LIN {X 0,Y 246.753,Z 542.174,A -85,B 0,C 180,E1 -19452.863,E2 -19452.863} C_VEL
LIN {X 0,Y 244.943,Z 545.036,A -85,B 0,C 180,E1 -19455.038,E2 -19455.038} C_VEL
LIN {X 0,Y 243.69,Z 547.692,A -85,B 0,C 180,E1 -19456.783,E2 -19456.783} C_VEL
LIN {X 0,Y 243.644,Z 549.387,A -85,B 0,C 180,E1 -19458.123,E2 -19458.123} C_VEL
LIN {X 0,Y 243.903,Z 549.825,A -85,B 0,C 180,E1 -19458.574,E2 -19458.574} C_VEL
LIN {X 0,Y 249.564,Z 556.197,A -85,B 0,C 180,E1 -19464.321,E2 -19464.321} C_VEL
LIN {X 0,Y 254.169,Z 562.573,A -85,B 0,C 180,E1 -19467.813,E2 -19467.813} C_VEL
LIN {X 0,Y 257.606,Z 568.633,A -85,B 0,C 180,E1 -19470.142,E2 -19470.142} C_VEL
LIN {X 0,Y 261.65,Z 575.949,A -85,B 0,C 180,E1 -19472.607,E2 -19472.607} C_VEL
LIN {X 0,Y 267.284,Z 587.342,A -85,B 0,C 180,E1 -19475.896,E2 -19475.896} C_VEL
LIN {X 0,Y 271.703,Z 597.971,A -85,B 0,C 180,E1 -19478.492,E2 -19478.492} C_VEL
LIN {X 0,Y 273.705,Z 604.625,A -85,B 0,C 180,E1 -19479.839,E2 -19479.839} C_VEL
LIN {X 0,Y 275.017,Z 618.379,A -85,B 0,C 180,E1 -19481.932,E2 -19481.932} C_VEL
LIN {X 0,Y 275.465,Z 630.728,A -85,B 0,C 180,E1 -19483.791,E2 -19483.791} C_VEL
LIN {X 0,Y 274.604,Z 645.683,A -85,B 0,C 180,E1 -19486.014,E2 -19486.014} C_VEL
LIN {X 0,Y 273.727,Z 654.542,A -85,B 0,C 180,E1 -19487.416,E2 -19487.416} C_VEL
LIN {X 0,Y 268.638,Z 668.348,A -85,B 0,C 180,E1 -19489.156,E2 -19489.156} C_VEL
LIN {X 0,Y 263.474,Z 681.321,A -85,B 0,C 180,E1 -19491.185,E2 -19491.185} C_VEL
LIN {X 0,Y 258.614,Z 692.426,A -85,B 0,C 180,E1 -19493.286,E2 -19493.286} C_VEL
LIN {X 0,Y 253.557,Z 703.587,A -85,B 0,C 180,E1 -19495.858,E2 -19495.858} C_VEL
LIN {X 0,Y 249.031,Z 713.236,A -85,B 0,C 180,E1 -19498.529,E2 -19498.529} C_VEL
LIN {X 0,Y 244.437,Z 722.628,A -85,B 0,C 180,E1 -19501.682,E2 -19501.682} C_VEL
LIN {X 0,Y 240.71,Z 730.545,A -85,B 0,C 180,E1 -19504.983,E2 -19504.983} C_VEL
LIN {X 0,Y 237.833,Z 737.107,A -85,B 0,C 180,E1 -19508.325,E2 -19508.325} C_VEL
LIN {X 0,Y 235.644,Z 742.544,A -85,B 0,C 180,E1 -19511.752,E2 -19511.752} C_VEL
LIN {X 0,Y 234.505,Z 745.925,A -85,B 0,C 180,E1 -19514.354,E2 -19514.354} C_VEL
LIN {X 0,Y 233.377,Z 749.429,A -85,B 0,C 180,E1 -19517.833,E2 -19517.833} C_VEL
LIN {X 0,Y 232.962,Z 752.026,A -85,B 0,C 180,E1 -19521.326,E2 -19521.326} C_VEL
LIN {X 0,Y 233.053,Z 753.553,A -85,B 0,C 180,E1 -19524.811,E2 -19524.811} C_VEL
LIN {X 0,Y 233.098,Z 754.168,A -85,B 0,C 180,E1 -19528.274,E2 -19528.274} C_VEL
LIN {X 0,Y 233.218,Z 754.054,A -85,B 0,C 180,E1 -19530.002,E2 -19530.002} C_VEL
LIN {X 0,Y 233.126,Z 753.085,A -85,B 0,C 180,E1 -19533.458,E2 -19533.458} C_VEL
LIN {X 0,Y 233.073,Z 751.097,A -85,B 0,C 180,E1 -19536.929,E2 -19536.929} C_VEL
LIN {X 0,Y 233.202,Z 747.994,A -85,B 0,C 180,E1 -19540.419,E2 -19540.419} C_VEL
LIN {X 0,Y 233.915,Z 743.858,A -85,B 0,C 180,E1 -19543.91,E2 -19543.91} C_VEL
LIN {X 0,Y 235.501,Z 736.962,A -85,B 0,C 180,E1 -19548.263,E2 -19548.263} C_VEL
LIN {X 0,Y 238.22,Z 728.654,A -85,B 0,C 180,E1 -19552.554,E2 -19552.554} C_VEL
LIN {X 0,Y 242.184,Z 720.832,A -85,B 0,C 180,E1 -19556.732,E2 -19556.732} C_VEL
LIN {X 0,Y 247.611,Z 711.66,A -85,B 0,C 180,E1 -19560.725,E2 -19560.725} C_VEL
LIN {X 0,Y 255.156,Z 700.072,A -85,B 0,C 180,E1 -19564.859,E2 -19564.859} C_VEL
LIN {X 0,Y 263.466,Z 688.242,A -85,B 0,C 180,E1 -19568.332,E2 -19568.332} C_VEL
LIN {X 0,Y 273.098,Z 675.378,A -85,B 0,C 180,E1 -19571.437,E2 -19571.437} C_VEL
LIN {X 0,Y 284.184,Z 661.013,A -85,B 0,C 180,E1 -19574.319,E2 -19574.319} C_VEL
LIN {X 0,Y 294.963,Z 646.585,A -85,B 0,C 180,E1 -19577.616,E2 -19577.616} C_VEL
LIN {X 0,Y 295.785,Z 645.371,A -85,B 0,C 180,E1 -19578.296,E2 -19578.296} C_VEL
LIN {X 0,Y 284.508,Z 656.676,A -85,B 0,C 180,E1 -19580.957,E2 -19580.957} C_VEL
LIN {X 0,Y 274.466,Z 666.622,A -85,B 0,C 180,E1 -19583.919,E2 -19583.919} C_VEL
LIN {X 0,Y 265.614,Z 675.208,A -85,B 0,C 180,E1 -19587.152,E2 -19587.152} C_VEL
LIN {X 0,Y 257.876,Z 682.625,A -85,B 0,C 180,E1 -19590.623,E2 -19590.623} C_VEL
LIN {X 0,Y 251.327,Z 688.726,A -85,B 0,C 180,E1 -19594.315,E2 -19594.315} C_VEL
LIN {X 0,Y 245.942,Z 693.539,A -85,B 0,C 180,E1 -19598.194,E2 -19598.194} C_VEL
LIN {X 0,Y 242.458,Z 696.492,A -85,B 0,C 180,E1 -19601.407,E2 -19601.407} C_VEL
LIN {X 0,Y 238.521,Z 699.293,A -85,B 0,C 180,E1 -19606.367,E2 -19606.367} C_VEL
LIN {X 0,Y 236.779,Z 700.073,A -85,B 0,C 180,E1 -19609.742,E2 -19609.742} C_VEL
LIN {X 0,Y 235.445,Z 700.059,A -85,B 0,C 180,E1 -19613.143,E2 -19613.143} C_VEL
LIN {X 0,Y 234.465,Z 699.144,A -85,B 0,C 180,E1 -19616.564,E2 -19616.564} C_VEL
LIN {X 0,Y 234.06,Z 697.294,A -85,B 0,C 180,E1 -19620.001,E2 -19620.001} C_VEL
LIN {X 0,Y 234.205,Z 694.494,A -85,B 0,C 180,E1 -19623.441,E2 -19623.441} C_VEL
LIN {X 0,Y 234.316,Z 690.68,A -85,B 0,C 180,E1 -19626.891,E2 -19626.891} C_VEL
LIN {X 0,Y 234.865,Z 685.837,A -85,B 0,C 180,E1 -19630.344,E2 -19630.344} C_VEL
LIN {X 0,Y 235.755,Z 679.792,A -85,B 0,C 180,E1 -19633.798,E2 -19633.798} C_VEL
LIN {X 0,Y 237.252,Z 672.466,A -85,B 0,C 180,E1 -19637.232,E2 -19637.232} C_VEL
LIN {X 0,Y 239.246,Z 663.732,A -85,B 0,C 180,E1 -19640.642,E2 -19640.642} C_VEL
LIN {X 0,Y 241.824,Z 653.381,A -85,B 0,C 180,E1 -19644.009,E2 -19644.009} C_VEL
LIN {X 0,Y 244.787,Z 641.972,A -85,B 0,C 180,E1 -19647.12,E2 -19647.12} C_VEL
LIN {X 0,Y 247.812,Z 630.51,A -85,B 0,C 180,E1 -19649.757,E2 -19649.757} C_VEL
LIN {X 0,Y 251.044,Z 618.323,A -85,B 0,C 180,E1 -19652.135,E2 -19652.135} C_VEL
LIN {X 0,Y 254.521,Z 604.23,A -85,B 0,C 180,E1 -19654.477,E2 -19654.477} C_VEL
LIN {X 0,Y 257.949,Z 589.052,A -85,B 0,C 180,E1 -19656.585,E2 -19656.585} C_VEL
LIN {X 0,Y 258.395,Z 586.367,A -85,B 0,C 180,E1 -19656.936,E2 -19656.936} C_VEL
LIN {X 0,Y 254.018,Z 573.751,A -85,B 0,C 180,E1 -19659.222,E2 -19659.222} C_VEL
LIN {X 0,Y 248.117,Z 558.525,A -85,B 0,C 180,E1 -19661.873,E2 -19661.873} C_VEL
LIN {X 0,Y 241.376,Z 543.393,A -85,B 0,C 180,E1 -19664.489,E2 -19664.489} C_VEL
LIN {X 0,Y 236.726,Z 534.301,A -85,B 0,C 180,E1 -19666.059,E2 -19666.059} C_VEL
LIN {X 0,Y 235.778,Z 532.761,A -85,B 0,C 180,E1 -19666.392,E2 -19666.392} C_VEL
LIN {X 0,Y 236.767,Z 536.937,A -85,B 0,C 180,E1 -19670.514,E2 -19670.514} C_VEL
LIN {X 0,Y 236.972,Z 538.218,A -85,B 0,C 180,E1 -19671.708,E2 -19671.708} C_VEL
LIN {X 0,Y 238.818,Z 541.601,A -85,B 0,C 180,E1 -19672.353,E2 -19672.353} C_VEL
LIN {X 0,Y 240.695,Z 543.935,A -85,B 0,C 180,E1 -19672.942,E2 -19672.942} C_VEL
LIN {X 0,Y 244.26,Z 549.567,A -85,B 0,C 180,E1 -19674.084,E2 -19674.084} C_VEL
LIN {X 0,Y 248.925,Z 556.937,A -85,B 0,C 180,E1 -19675.567,E2 -19675.567} C_VEL
LIN {X 0,Y 255.974,Z 570.468,A -85,B 0,C 180,E1 -19678.026,E2 -19678.026} C_VEL
LIN {X 0,Y 260.019,Z 580.879,A -85,B 0,C 180,E1 -19679.709,E2 -19679.709} C_VEL
LIN {X 0,Y 264.07,Z 594.759,A -85,B 0,C 180,E1 -19681.87,E2 -19681.87} C_VEL
LIN {X 0,Y 266.896,Z 606.997,A -85,B 0,C 180,E1 -19683.819,E2 -19683.819} C_VEL
LIN {X 0,Y 267.602,Z 611.223,A -85,B 0,C 180,E1 -19684.504,E2 -19684.504} C_VEL
LIN {X 0,Y 264.738,Z 624.004,A -85,B 0,C 180,E1 -19685.909,E2 -19685.909} C_VEL
LIN {X 0,Y 260.749,Z 638.524,A -85,B 0,C 180,E1 -19687.829,E2 -19687.829} C_VEL
LIN {X 0,Y 256.639,Z 651.83,A -85,B 0,C 180,E1 -19689.981,E2 -19689.981} C_VEL
LIN {X 0,Y 252.939,Z 663.185,A -85,B 0,C 180,E1 -19692.202,E2 -19692.202} C_VEL
LIN {X 0,Y 249.018,Z 674.563,A -85,B 0,C 180,E1 -19694.865,E2 -19694.865} C_VEL
LIN {X 0,Y 244.972,Z 685.564,A -85,B 0,C 180,E1 -19697.993,E2 -19697.993} C_VEL
LIN {X 0,Y 242.016,Z 693.828,A -85,B 0,C 180,E1 -19700.878,E2 -19700.878} C_VEL
LIN {X 0,Y 239.165,Z 701.547,A -85,B 0,C 180,E1 -19704.095,E2 -19704.095} C_VEL
LIN {X 0,Y 236.935,Z 708.138,A -85,B 0,C 180,E1 -19707.448,E2 -19707.448} C_VEL
LIN {X 0,Y 234.863,Z 714.656,A -85,B 0,C 180,E1 -19711.713,E2 -19711.713} C_VEL
LIN {X 0,Y 233.843,Z 718.603,A -85,B 0,C 180,E1 -19715.171,E2 -19715.171} C_VEL
LIN {X 0,Y 233.175,Z 721.586,A -85,B 0,C 180,E1 -19718.666,E2 -19718.666} C_VEL
LIN {X 0,Y 232.819,Z 723.564,A -85,B 0,C 180,E1 -19722.197,E2 -19722.197} C_VEL
LIN {X 0,Y 232.769,Z 724.563,A -85,B 0,C 180,E1 -19725.766,E2 -19725.766} C_VEL
LIN {X 0,Y 233.009,Z 724.613,A -85,B 0,C 180,E1 -19729.375,E2 -19729.375} C_VEL
LIN {X 0,Y 233.618,Z 723.592,A -85,B 0,C 180,E1 -19733.02,E2 -19733.02} C_VEL
LIN {X 0,Y 234.77,Z 721.586,A -85,B 0,C 180,E1 -19736.679,E2 -19736.679} C_VEL
LIN {X 0,Y 236.558,Z 718.256,A -85,B 0,C 180,E1 -19740.505,E2 -19740.505} C_VEL
LIN {X 0,Y 238.815,Z 714.066,A -85,B 0,C 180,E1 -19743.994,E2 -19743.994} C_VEL
LIN {X 0,Y 241.917,Z 708.476,A -85,B 0,C 180,E1 -19747.592,E2 -19747.592} C_VEL
LIN {X 0,Y 245.817,Z 701.452,A -85,B 0,C 180,E1 -19751.112,E2 -19751.112} C_VEL
LIN {X 0,Y 250.527,Z 692.801,A -85,B 0,C 180,E1 -19754.53,E2 -19754.53} C_VEL
LIN {X 0,Y 255.281,Z 683.712,A -85,B 0,C 180,E1 -19757.426,E2 -19757.426} C_VEL
LIN {X 0,Y 260.584,Z 672.958,A -85,B 0,C 180,E1 -19760.229,E2 -19760.229} C_VEL
LIN {X 0,Y 266.019,Z 661.133,A -85,B 0,C 180,E1 -19762.735,E2 -19762.735} C_VEL
LIN {X 0,Y 270.921,Z 649.417,A -85,B 0,C 180,E1 -19764.781,E2 -19764.781} C_VEL
LIN {X 0,Y 276.221,Z 635.397,A -85,B 0,C 180,E1 -19766.763,E2 -19766.763} C_VEL
LIN {X 0,Y 280.705,Z 621.712,A -85,B 0,C 180,E1 -19768.345,E2 -19768.345} C_VEL
LIN {X 0,Y 280.523,Z 617.811,A -85,B 0,C 180,E1 -19769.095,E2 -19769.095} C_VEL
LIN {X 0,Y 278.114,Z 605.638,A -85,B 0,C 180,E1 -19771.717,E2 -19771.717} C_VEL
LIN {X 0,Y 275.799,Z 598.13,A -85,B 0,C 180,E1 -19773.516,E2 -19773.516} C_VEL
LIN {X 0,Y 271.396,Z 587.981,A -85,B 0,C 180,E1 -19776.335,E2 -19776.335} C_VEL
LIN {X 0,Y 267.044,Z 579.471,A -85,B 0,C 180,E1 -19778.986,E2 -19778.986} C_VEL
LIN {X 0,Y 263.885,Z 574.325,A -85,B 0,C 180,E1 -19780.857,E2 -19780.857} C_VEL
LIN {X 0,Y 261.135,Z 569.949,A -85,B 0,C 180,E1 -19782.577,E2 -19782.577} C_VEL
LIN {X 0,Y 258.457,Z 565.967,A -85,B 0,C 180,E1 -19784.271,E2 -19784.271} C_VEL
LIN {X 0,Y 255.085,Z 561.378,A -85,B 0,C 180,E1 -19786.557,E2 -19786.557} C_VEL
LIN {X 0,Y 254.143,Z 560.119,A -85,B 0,C 180,E1 -19787.218,E2 -19787.218} C_VEL
LIN {X 0,Y 251.125,Z 556.561,A -85,B 0,C 180,E1 -19789.467,E2 -19789.467} C_VEL
LIN {X 0,Y 250.177,Z 554.992,A -85,B 0,C 180,E1 -19790.296,E2 -19790.296} C_VEL
LIN {X 0,Y 246.659,Z 551.307,A -85,B 0,C 180,E1 -19793.455,E2 -19793.455} C_VEL
LIN {X 0,Y 245.575,Z 549.621,A -85,B 0,C 180,E1 -19794.662,E2 -19794.662} C_VEL
LIN {X 0,Y 240.898,Z 544.483,A -85,B 0,C 180,E1 -19802.194,E2 -19802.194} C_VEL
LIN {X 0,Y 241.02,Z 544.658,A -85,B 0,C 180,E1 -19807.53,E2 -19807.53} C_VEL
LIN {X 0,Y 241.423,Z 545.578,A -85,B 0,C 180,E1 -19811.757,E2 -19811.757} C_VEL
LIN {X 0,Y 242.13,Z 546.869,A -85,B 0,C 180,E1 -19815.142,E2 -19815.142} C_VEL
LIN {X 0,Y 242.607,Z 547.879,A -85,B 0,C 180,E1 -19816.629,E2 -19816.629} C_VEL
LIN {X 0,Y 243.903,Z 549.825,A -85,B 0,C 180,E1 -19818.574,E2 -19818.574} C_VEL
LIN {X 0,Y 244.879,Z 551.629,A -85,B 0,C 180,E1 -19819.87,E2 -19819.87} C_VEL
LIN {X 0,Y 246.399,Z 556.445,A -85,B 0,C 180,E1 -19821.853,E2 -19821.853} C_VEL
LIN {X 0,Y 247.704,Z 560.852,A -85,B 0,C 180,E1 -19823.38,E2 -19823.38} C_VEL
LIN {X 0,Y 249.325,Z 564.702,A -85,B 0,C 180,E1 -19824.955,E2 -19824.955} C_VEL
LIN {X 0,Y 252.237,Z 569.047,A -85,B 0,C 180,E1 -19827.267,E2 -19827.267} C_VEL
LIN {X 0,Y 256.292,Z 576.683,A -85,B 0,C 180,E1 -19830.199,E2 -19830.199} C_VEL
LIN {X 0,Y 258.961,Z 581.967,A -85,B 0,C 180,E1 -19832.009,E2 -19832.009} C_VEL
LIN {X 0,Y 264.002,Z 592.929,A -85,B 0,C 180,E1 -19835.27,E2 -19835.27} C_VEL
LIN {X 0,Y 267.828,Z 603.023,A -85,B 0,C 180,E1 -19837.809,E2 -19837.809} C_VEL
LIN {X 0,Y 269.334,Z 608.443,A -85,B 0,C 180,E1 -19838.979,E2 -19838.979} C_VEL
LIN {X 0,Y 270.277,Z 621.61,A -85,B 0,C 180,E1 -19841.058,E2 -19841.058} C_VEL
LIN {X 0,Y 270.324,Z 634.577,A -85,B 0,C 180,E1 -19843.092,E2 -19843.092} C_VEL
LIN {X 0,Y 269.048,Z 649.765,A -85,B 0,C 180,E1 -19845.451,E2 -19845.451} C_VEL
LIN {X 0,Y 268.079,Z 656.629,A -85,B 0,C 180,E1 -19846.567,E2 -19846.567} C_VEL
LIN {X 0,Y 262.85,Z 669.944,A -85,B 0,C 180,E1 -19848.317,E2 -19848.317} C_VEL
LIN {X 0,Y 257.961,Z 681.592,A -85,B 0,C 180,E1 -19850.193,E2 -19850.193} C_VEL
LIN {X 0,Y 252.932,Z 692.633,A -85,B 0,C 180,E1 -19852.319,E2 -19852.319} C_VEL
LIN {X 0,Y 247.653,Z 703.683,A -85,B 0,C 180,E1 -19854.927,E2 -19854.927} C_VEL
LIN {X 0,Y 242.915,Z 713.226,A -85,B 0,C 180,E1 -19857.642,E2 -19857.642} C_VEL
LIN {X 0,Y 238.131,Z 722.555,A -85,B 0,C 180,E1 -19860.861,E2 -19860.861} C_VEL
LIN {X 0,Y 234.26,Z 730.24,A -85,B 0,C 180,E1 -19864.16,E2 -19864.16} C_VEL
LIN {X 0,Y 231.134,Z 736.895,A -85,B 0,C 180,E1 -19867.664,E2 -19867.664} C_VEL
LIN {X 0,Y 228.788,Z 742.299,A -85,B 0,C 180,E1 -19871.185,E2 -19871.185} C_VEL
LIN {X 0,Y 227.569,Z 745.625,A -85,B 0,C 180,E1 -19873.864,E2 -19873.864} C_VEL
LIN {X 0,Y 226.364,Z 749.09,A -85,B 0,C 180,E1 -19877.45,E2 -19877.45} C_VEL
LIN {X 0,Y 225.891,Z 751.636,A -85,B 0,C 180,E1 -19881.053,E2 -19881.053} C_VEL
LIN {X 0,Y 225.987,Z 753.139,A -85,B 0,C 180,E1 -19884.649,E2 -19884.649} C_VEL
LIN {X 0,Y 226.021,Z 753.704,A -85,B 0,C 180,E1 -19888.22,E2 -19888.22} C_VEL
LIN {X 0,Y 226.134,Z 753.589,A -85,B 0,C 180,E1 -19890.002,E2 -19890.002} C_VEL
LIN {X 0,Y 226.06,Z 752.568,A -85,B 0,C 180,E1 -19893.567,E2 -19893.567} C_VEL
LIN {X 0,Y 226.05,Z 751.42,A -85,B 0,C 180,E1 -19895.8,E2 -19895.8} C_VEL
LIN {X 0,Y 225.986,Z 749.093,A -85,B 0,C 180,E1 -19898.947,E2 -19898.947} C_VEL
LIN {X 0,Y 226.701,Z 744.331,A -85,B 0,C 180,E1 -19903.447,E2 -19903.447} C_VEL
LIN {X 0,Y 227.817,Z 739.299,A -85,B 0,C 180,E1 -19906.998,E2 -19906.998} C_VEL
LIN {X 0,Y 229.659,Z 732.91,A -85,B 0,C 180,E1 -19910.607,E2 -19910.607} C_VEL
LIN {X 0,Y 230.878,Z 729.9,A -85,B 0,C 180,E1 -19912.367,E2 -19912.367} C_VEL
LIN {X 0,Y 234.831,Z 722.594,A -85,B 0,C 180,E1 -19916.676,E2 -19916.676} C_VEL
LIN {X 0,Y 240.264,Z 714.068,A -85,B 0,C 180,E1 -19920.792,E2 -19920.792} C_VEL
LIN {X 0,Y 248.656,Z 702.21,A -85,B 0,C 180,E1 -19925.411,E2 -19925.411} C_VEL
LIN {X 0,Y 258.106,Z 689.925,A -85,B 0,C 180,E1 -19929.279,E2 -19929.279} C_VEL
LIN {X 0,Y 268.204,Z 677.514,A -85,B 0,C 180,E1 -19932.436,E2 -19932.436} C_VEL
LIN {X 0,Y 279.784,Z 663.808,A -85,B 0,C 180,E1 -19935.305,E2 -19935.305} C_VEL
LIN {X 0,Y 287.896,Z 653.936,A -85,B 0,C 180,E1 -19937.692,E2 -19937.692} C_VEL
LIN {X 0,Y 288.836,Z 652.749,A -85,B 0,C 180,E1 -19938.097,E2 -19938.097} C_VEL
LIN {X 0,Y 279.89,Z 660.96,A -85,B 0,C 180,E1 -19940.187,E2 -19940.187} C_VEL
LIN {X 0,Y 269.468,Z 670.219,A -85,B 0,C 180,E1 -19943.141,E2 -19943.141} C_VEL
LIN {X 0,Y 260.249,Z 678.331,A -85,B 0,C 180,E1 -19946.386,E2 -19946.386} C_VEL
LIN {X 0,Y 251.327,Z 685.932,A -85,B 0,C 180,E1 -19950.29,E2 -19950.29} C_VEL
LIN {X 0,Y 244.038,Z 691.945,A -85,B 0,C 180,E1 -19954.407,E2 -19954.407} C_VEL
LIN {X 0,Y 239.597,Z 695.402,A -85,B 0,C 180,E1 -19957.585,E2 -19957.585} C_VEL
LIN {X 0,Y 234.362,Z 699.158,A -85,B 0,C 180,E1 -19962.551,E2 -19962.551} C_VEL
LIN {X 0,Y 230.697,Z 701.035,A -85,B 0,C 180,E1 -19967.688,E2 -19967.688} C_VEL
LIN {X 0,Y 229.157,Z 701.206,A -85,B 0,C 180,E1 -19971.18,E2 -19971.18} C_VEL
LIN {X 0,Y 227.89,Z 700.597,A -85,B 0,C 180,E1 -19974.692,E2 -19974.692} C_VEL
LIN {X 0,Y 227.146,Z 699.046,A -85,B 0,C 180,E1 -19978.228,E2 -19978.228} C_VEL
LIN {X 0,Y 226.978,Z 696.569,A -85,B 0,C 180,E1 -19981.775,E2 -19981.775} C_VEL
LIN {X 0,Y 227.148,Z 694.987,A -85,B 0,C 180,E1 -19983.549,E2 -19983.549} C_VEL
LIN {X 0,Y 227.393,Z 689.847,A -85,B 0,C 180,E1 -19988.031,E2 -19988.031} C_VEL
LIN {X 0,Y 228.051,Z 684.536,A -85,B 0,C 180,E1 -19991.556,E2 -19991.556} C_VEL
LIN {X 0,Y 229.106,Z 678.017,A -85,B 0,C 180,E1 -19995.115,E2 -19995.115} C_VEL
LIN {X 0,Y 231.133,Z 669.112,A -85,B 0,C 180,E1 -19999.08,E2 -19999.08} C_VEL
LIN {X 0,Y 233.46,Z 659.623,A -85,B 0,C 180,E1 -20002.571,E2 -20002.571} C_VEL
LIN {X 0,Y 236.473,Z 648.366,A -85,B 0,C 180,E1 -20006.001,E2 -20006.001} C_VEL
LIN {X 0,Y 239.467,Z 636.847,A -85,B 0,C 180,E1 -20008.964,E2 -20008.964} C_VEL
LIN {X 0,Y 243.428,Z 622.376,A -85,B 0,C 180,E1 -20012.04,E2 -20012.04} C_VEL
LIN {X 0,Y 247.261,Z 607.618,A -85,B 0,C 180,E1 -20014.644,E2 -20014.644} C_VEL
LIN {X 0,Y 250.722,Z 593.093,A -85,B 0,C 180,E1 -20016.793,E2 -20016.793} C_VEL
LIN {X 0,Y 251.718,Z 588.719,A -85,B 0,C 180,E1 -20017.357,E2 -20017.357} C_VEL
LIN {X 0,Y 248.934,Z 579.925,A -85,B 0,C 180,E1 -20019.001,E2 -20019.001} C_VEL
LIN {X 0,Y 243.897,Z 566.294,A -85,B 0,C 180,E1 -20021.511,E2 -20021.511} C_VEL
LIN {X 0,Y 238.559,Z 553.457,A -85,B 0,C 180,E1 -20023.828,E2 -20023.828} C_VEL
LIN {X 0,Y 232.811,Z 541.092,A -85,B 0,C 180,E1 -20026.025,E2 -20026.025} C_VEL
LIN {X 0,Y 231.778,Z 539.224,A -85,B 0,C 180,E1 -20026.382,E2 -20026.382} C_VEL
LIN {X 0,Y 229.341,Z 536.139,A -85,B 0,C 180,E1 -20027.108,E2 -20027.108} C_VEL
LIN {X 0,Y 229.987,Z 538.855,A -85,B 0,C 180,E1 -20029.761,E2 -20029.761} C_VEL
LIN {X 0,Y 231.969,Z 542.273,A -85,B 0,C 180,E1 -20030.504,E2 -20030.504} C_VEL
LIN {X 0,Y 233.725,Z 544.503,A -85,B 0,C 180,E1 -20031.105,E2 -20031.105} C_VEL
LIN {X 0,Y 236.203,Z 548.126,A -85,B 0,C 180,E1 -20031.955,E2 -20031.955} C_VEL
LIN {X 0,Y 240.849,Z 555.572,A -85,B 0,C 180,E1 -20033.567,E2 -20033.567} C_VEL
LIN {X 0,Y 244.842,Z 562.201,A -85,B 0,C 180,E1 -20034.963,E2 -20034.963} C_VEL
LIN {X 0,Y 251.239,Z 574.914,A -85,B 0,C 180,E1 -20037.378,E2 -20037.378} C_VEL
LIN {X 0,Y 254.863,Z 584.868,A -85,B 0,C 180,E1 -20039.066,E2 -20039.066} C_VEL
LIN {X 0,Y 258.336,Z 597.372,A -85,B 0,C 180,E1 -20041.118,E2 -20041.118} C_VEL
LIN {X 0,Y 261.142,Z 610.44,A -85,B 0,C 180,E1 -20043.299,E2 -20043.299} C_VEL
LIN {X 0,Y 261.479,Z 613.997,A -85,B 0,C 180,E1 -20043.861,E2 -20043.861} C_VEL
LIN {X 0,Y 257.585,Z 629.196,A -85,B 0,C 180,E1 -20045.626,E2 -20045.626} C_VEL
LIN {X 0,Y 253.592,Z 642.956,A -85,B 0,C 180,E1 -20047.599,E2 -20047.599} C_VEL
LIN {X 0,Y 249.426,Z 655.715,A -85,B 0,C 180,E1 -20049.807,E2 -20049.807} C_VEL
LIN {X 0,Y 245.089,Z 668.293,A -85,B 0,C 180,E1 -20052.475,E2 -20052.475} C_VEL
LIN {X 0,Y 241.15,Z 678.936,A -85,B 0,C 180,E1 -20055.224,E2 -20055.224} C_VEL
LIN {X 0,Y 237.619,Z 688.069,A -85,B 0,C 180,E1 -20058.05,E2 -20058.05} C_VEL
LIN {X 0,Y 234.303,Z 696.949,A -85,B 0,C 180,E1 -20061.373,E2 -20061.373} C_VEL
LIN {X 0,Y 231.512,Z 704.4,A -85,B 0,C 180,E1 -20064.773,E2 -20064.773} C_VEL
LIN {X 0,Y 228.911,Z 711.887,A -85,B 0,C 180,E1 -20069.119,E2 -20069.119} C_VEL
LIN {X 0,Y 227.22,Z 717.586,A -85,B 0,C 180,E1 -20073.545,E2 -20073.545} C_VEL
LIN {X 0,Y 226.329,Z 720.926,A -85,B 0,C 180,E1 -20077.133,E2 -20077.133} C_VEL
LIN {X 0,Y 225.841,Z 723.338,A -85,B 0,C 180,E1 -20080.759,E2 -20080.759} C_VEL
LIN {X 0,Y 225.719,Z 724.719,A -85,B 0,C 180,E1 -20084.421,E2 -20084.421} C_VEL
LIN {X 0,Y 225.791,Z 725.161,A -85,B 0,C 180,E1 -20088.133,E2 -20088.133} C_VEL
LIN {X 0,Y 226.312,Z 724.602,A -85,B 0,C 180,E1 -20091.877,E2 -20091.877} C_VEL
LIN {X 0,Y 227.584,Z 722.53,A -85,B 0,C 180,E1 -20096.419,E2 -20096.419} C_VEL
LIN {X 0,Y 228.872,Z 720.333,A -85,B 0,C 180,E1 -20099.424,E2 -20099.424} C_VEL
LIN {X 0,Y 231.073,Z 716.46,A -85,B 0,C 180,E1 -20103.191,E2 -20103.191} C_VEL
LIN {X 0,Y 234.065,Z 711.37,A -85,B 0,C 180,E1 -20106.904,E2 -20106.904} C_VEL
LIN {X 0,Y 237.837,Z 704.962,A -85,B 0,C 180,E1 -20110.546,E2 -20110.546} C_VEL
LIN {X 0,Y 242.491,Z 697.048,A -85,B 0,C 180,E1 -20114.07,E2 -20114.07} C_VEL
LIN {X 0,Y 246.907,Z 689.104,A -85,B 0,C 180,E1 -20116.909,E2 -20116.909} C_VEL
LIN {X 0,Y 252.097,Z 679.363,A -85,B 0,C 180,E1 -20119.782,E2 -20119.782} C_VEL
LIN {X 0,Y 257.458,Z 668.759,A -85,B 0,C 180,E1 -20122.335,E2 -20122.335} C_VEL
LIN {X 0,Y 263.296,Z 656.07,A -85,B 0,C 180,E1 -20124.827,E2 -20124.827} C_VEL
LIN {X 0,Y 268.592,Z 643.28,A -85,B 0,C 180,E1 -20126.854,E2 -20126.854} C_VEL
LIN {X 0,Y 273.289,Z 630.509,A -85,B 0,C 180,E1 -20128.516,E2 -20128.516} C_VEL
LIN {X 0,Y 275.539,Z 623.513,A -85,B 0,C 180,E1 -20129.327,E2 -20129.327} C_VEL
LIN {X 0,Y 274.313,Z 614.64,A -85,B 0,C 180,E1 -20131.289,E2 -20131.289} C_VEL
LIN {X 0,Y 272.564,Z 606.596,A -85,B 0,C 180,E1 -20133.176,E2 -20133.176} C_VEL
LIN {X 0,Y 270.258,Z 599.732,A -85,B 0,C 180,E1 -20135.002,E2 -20135.002} C_VEL
LIN {X 0,Y 265.598,Z 588.977,A -85,B 0,C 180,E1 -20138.256,E2 -20138.256} C_VEL
LIN {X 0,Y 261.078,Z 580.613,A -85,B 0,C 180,E1 -20141.255,E2 -20141.255} C_VEL
LIN {X 0,Y 258.197,Z 575.889,A -85,B 0,C 180,E1 -20143.189,E2 -20143.189} C_VEL
LIN {X 0,Y 255.333,Z 571.346,A -85,B 0,C 180,E1 -20145.249,E2 -20145.249} C_VEL
LIN {X 0,Y 252.671,Z 567.345,A -85,B 0,C 180,E1 -20147.232,E2 -20147.232} C_VEL
LIN {X 0,Y 249.307,Z 563.057,A -85,B 0,C 180,E1 -20149.973,E2 -20149.973} C_VEL
LIN {X 0,Y 248.375,Z 561.59,A -85,B 0,C 180,E1 -20150.817,E2 -20150.817} C_VEL
LIN {X 0,Y 245.096,Z 557.788,A -85,B 0,C 180,E1 -20154.033,E2 -20154.033} C_VEL
LIN {X 0,Y 244.274,Z 556.481,A -85,B 0,C 180,E1 -20155.048,E2 -20155.048} C_VEL
LIN {X 0,Y 240.008,Z 551.587,A -85,B 0,C 180,E1 -20162.097,E2 -20162.097} C_VEL
LIN {X 0,Y 238.942,Z 551.538,A -85,B 0,C 180,E1 -20168.456,E2 -20168.456} C_VEL
LIN {X 0,Y 240.291,Z 553.311,A -85,B 0,C 180,E1 -20173.962,E2 -20173.962} C_VEL
LIN {X 0,Y 241.497,Z 554.757,A -85,B 0,C 180,E1 -20176.306,E2 -20176.306} C_VEL
LIN {X 0,Y 247.891,Z 562.589,A -85,B 0,C 180,E1 -20183.717,E2 -20183.717} C_VEL
LIN {X 0,Y 249.325,Z 564.702,A -85,B 0,C 180,E1 -20184.955,E2 -20184.955} C_VEL
LIN {X 0,Y 250.169,Z 566.638,A -85,B 0,C 180,E1 -20185.721,E2 -20185.721} C_VEL
LIN {X 0,Y 251.47,Z 571.825,A -85,B 0,C 180,E1 -20187.067,E2 -20187.067} C_VEL
LIN {X 0,Y 253.45,Z 581.689,A -85,B 0,C 180,E1 -20189.28,E2 -20189.28} C_VEL
LIN {X 0,Y 254.807,Z 584.881,A -85,B 0,C 180,E1 -20190.368,E2 -20190.368} C_VEL
LIN {X 0,Y 258.01,Z 592.18,A -85,B 0,C 180,E1 -20192.762,E2 -20192.762} C_VEL
LIN {X 0,Y 261.56,Z 601.034,A -85,B 0,C 180,E1 -20195.347,E2 -20195.347} C_VEL
LIN {X 0,Y 263.973,Z 608.509,A -85,B 0,C 180,E1 -20197.231,E2 -20197.231} C_VEL
LIN {X 0,Y 265.034,Z 612.903,A -85,B 0,C 180,E1 -20198.193,E2 -20198.193} C_VEL
LIN {X 0,Y 265.543,Z 627.387,A -85,B 0,C 180,E1 -20200.592,E2 -20200.592} C_VEL
LIN {X 0,Y 265.149,Z 638.527,A -85,B 0,C 180,E1 -20202.394,E2 -20202.394} C_VEL
LIN {X 0,Y 263.389,Z 653.939,A -85,B 0,C 180,E1 -20204.927,E2 -20204.927} C_VEL
LIN {X 0,Y 262.515,Z 658.448,A -85,B 0,C 180,E1 -20205.661,E2 -20205.661} C_VEL
LIN {X 0,Y 257.029,Z 671.802,A -85,B 0,C 180,E1 -20207.474,E2 -20207.474} C_VEL
LIN {X 0,Y 251.66,Z 683.813,A -85,B 0,C 180,E1 -20209.515,E2 -20209.515} C_VEL
LIN {X 0,Y 245.66,Z 696.098,A -85,B 0,C 180,E1 -20212.045,E2 -20212.045} C_VEL
LIN {X 0,Y 239.746,Z 707.725,A -85,B 0,C 180,E1 -20215.037,E2 -20215.037} C_VEL
LIN {X 0,Y 234.279,Z 718.041,A -85,B 0,C 180,E1 -20218.336,E2 -20218.336} C_VEL
LIN {X 0,Y 229.717,Z 726.533,A -85,B 0,C 180,E1 -20221.695,E2 -20221.695} C_VEL
LIN {X 0,Y 225.997,Z 733.594,A -85,B 0,C 180,E1 -20225.179,E2 -20225.179} C_VEL
LIN {X 0,Y 223.102,Z 739.506,A -85,B 0,C 180,E1 -20228.763,E2 -20228.763} C_VEL
LIN {X 0,Y 220.944,Z 744.494,A -85,B 0,C 180,E1 -20232.603,E2 -20232.603} C_VEL
LIN {X 0,Y 219.932,Z 747.183,A -85,B 0,C 180,E1 -20235.191,E2 -20235.191} C_VEL
LIN {X 0,Y 219.005,Z 750.111,A -85,B 0,C 180,E1 -20238.901,E2 -20238.901} C_VEL
LIN {X 0,Y 218.8,Z 752.127,A -85,B 0,C 180,E1 -20242.62,E2 -20242.62} C_VEL
LIN {X 0,Y 218.922,Z 752.725,A -85,B 0,C 180,E1 -20244.475,E2 -20244.475} C_VEL
LIN {X 0,Y 218.946,Z 753.239,A -85,B 0,C 180,E1 -20248.163,E2 -20248.163} C_VEL
LIN {X 0,Y 219.053,Z 753.124,A -85,B 0,C 180,E1 -20250.002,E2 -20250.002} C_VEL
LIN {X 0,Y 218.973,Z 752.05,A -85,B 0,C 180,E1 -20253.682,E2 -20253.682} C_VEL
LIN {X 0,Y 218.904,Z 750.002,A -85,B 0,C 180,E1 -20257.38,E2 -20257.38} C_VEL
LIN {X 0,Y 219.107,Z 746.786,A -85,B 0,C 180,E1 -20261.098,E2 -20261.098} C_VEL
LIN {X 0,Y 219.935,Z 742.536,A -85,B 0,C 180,E1 -20264.813,E2 -20264.813} C_VEL
LIN {X 0,Y 221.355,Z 737.054,A -85,B 0,C 180,E1 -20268.514,E2 -20268.514} C_VEL
LIN {X 0,Y 222.906,Z 732.217,A -85,B 0,C 180,E1 -20271.261,E2 -20271.261} C_VEL
LIN {X 0,Y 226.919,Z 725.12,A -85,B 0,C 180,E1 -20276.083,E2 -20276.083} C_VEL
LIN {X 0,Y 231.689,Z 718,A -85,B 0,C 180,E1 -20280.035,E2 -20280.035} C_VEL
LIN {X 0,Y 238.319,Z 709.097,A -85,B 0,C 180,E1 -20284.079,E2 -20284.079} C_VEL
LIN {X 0,Y 248.081,Z 697.027,A -85,B 0,C 180,E1 -20288.555,E2 -20288.555} C_VEL
LIN {X 0,Y 257.851,Z 685.833,A -85,B 0,C 180,E1 -20291.897,E2 -20291.897} C_VEL
LIN {X 0,Y 269.023,Z 673.637,A -85,B 0,C 180,E1 -20294.859,E2 -20294.859} C_VEL
LIN {X 0,Y 275.257,Z 666.908,A -85,B 0,C 180,E1 -20296.266,E2 -20296.266} C_VEL
LIN {X 0,Y 280.265,Z 661.311,A -85,B 0,C 180,E1 -20297.712,E2 -20297.712} C_VEL
LIN {X 0,Y 280.694,Z 660.659,A -85,B 0,C 180,E1 -20298.113,E2 -20298.113} C_VEL
LIN {X 0,Y 268.661,Z 670.474,A -85,B 0,C 180,E1 -20301.111,E2 -20301.111} C_VEL
LIN {X 0,Y 256.733,Z 679.981,A -85,B 0,C 180,E1 -20304.91,E2 -20304.91} C_VEL
LIN {X 0,Y 247.685,Z 686.922,A -85,B 0,C 180,E1 -20308.553,E2 -20308.553} C_VEL
LIN {X 0,Y 240.612,Z 692.174,A -85,B 0,C 180,E1 -20312.139,E2 -20312.139} C_VEL
LIN {X 0,Y 233.292,Z 697.323,A -85,B 0,C 180,E1 -20316.945,E2 -20316.945} C_VEL
LIN {X 0,Y 227.744,Z 700.665,A -85,B 0,C 180,E1 -20322.026,E2 -20322.026} C_VEL
LIN {X 0,Y 224.872,Z 701.945,A -85,B 0,C 180,E1 -20325.667,E2 -20325.667} C_VEL
LIN {X 0,Y 222.995,Z 702.35,A -85,B 0,C 180,E1 -20329.101,E2 -20329.101} C_VEL
LIN {X 0,Y 221.505,Z 701.943,A -85,B 0,C 180,E1 -20332.71,E2 -20332.71} C_VEL
LIN {X 0,Y 220.407,Z 700.709,A -85,B 0,C 180,E1 -20336.344,E2 -20336.344} C_VEL
LIN {X 0,Y 219.926,Z 698.519,A -85,B 0,C 180,E1 -20340.001,E2 -20340.001} C_VEL
LIN {X 0,Y 220.091,Z 695.403,A -85,B 0,C 180,E1 -20343.662,E2 -20343.662} C_VEL
LIN {X 0,Y 220.223,Z 691.3,A -85,B 0,C 180,E1 -20347.335,E2 -20347.335} C_VEL
LIN {X 0,Y 220.826,Z 686.082,A -85,B 0,C 180,E1 -20351.009,E2 -20351.009} C_VEL
LIN {X 0,Y 221.868,Z 679.733,A -85,B 0,C 180,E1 -20354.68,E2 -20354.68} C_VEL
LIN {X 0,Y 223.517,Z 672.061,A -85,B 0,C 180,E1 -20358.327,E2 -20358.327} C_VEL
LIN {X 0,Y 225.796,Z 662.898,A -85,B 0,C 180,E1 -20361.933,E2 -20361.933} C_VEL
LIN {X 0,Y 228.717,Z 652.104,A -85,B 0,C 180,E1 -20365.481,E2 -20365.481} C_VEL
LIN {X 0,Y 231.633,Z 641.292,A -85,B 0,C 180,E1 -20368.48,E2 -20368.48} C_VEL
LIN {X 0,Y 235.285,Z 628.248,A -85,B 0,C 180,E1 -20371.516,E2 -20371.516} C_VEL
LIN {X 0,Y 239.145,Z 614.079,A -85,B 0,C 180,E1 -20374.26,E2 -20374.26} C_VEL
LIN {X 0,Y 242.943,Z 599.386,A -85,B 0,C 180,E1 -20376.631,E2 -20376.631} C_VEL
LIN {X 0,Y 244.953,Z 590.68,A -85,B 0,C 180,E1 -20377.858,E2 -20377.858} C_VEL
LIN {X 0,Y 244.008,Z 586.721,A -85,B 0,C 180,E1 -20378.61,E2 -20378.61} C_VEL
LIN {X 0,Y 238.953,Z 572.48,A -85,B 0,C 180,E1 -20381.376,E2 -20381.376} C_VEL
LIN {X 0,Y 233.296,Z 558.469,A -85,B 0,C 180,E1 -20384.007,E2 -20384.007} C_VEL
LIN {X 0,Y 227.301,Z 545.09,A -85,B 0,C 180,E1 -20386.53,E2 -20386.53} C_VEL
LIN {X 0,Y 223.29,Z 540.218,A -85,B 0,C 180,E1 -20387.714,E2 -20387.714} C_VEL
LIN {X 0,Y 225.696,Z 543.664,A -85,B 0,C 180,E1 -20388.693,E2 -20388.693} C_VEL
LIN {X 0,Y 226.883,Z 545.125,A -85,B 0,C 180,E1 -20389.135,E2 -20389.135} C_VEL
LIN {X 0,Y 229.726,Z 549.174,A -85,B 0,C 180,E1 -20390.189,E2 -20390.189} C_VEL
LIN {X 0,Y 232.781,Z 553.813,A -85,B 0,C 180,E1 -20391.33,E2 -20391.33} C_VEL
LIN {X 0,Y 239.662,Z 565.39,A -85,B 0,C 180,E1 -20393.925,E2 -20393.925} C_VEL
LIN {X 0,Y 245.824,Z 577.972,A -85,B 0,C 180,E1 -20396.468,E2 -20396.468} C_VEL
LIN {X 0,Y 249.148,Z 586.953,A -85,B 0,C 180,E1 -20398.104,E2 -20398.104} C_VEL
LIN {X 0,Y 252.313,Z 598.405,A -85,B 0,C 180,E1 -20400.075,E2 -20400.075} C_VEL
LIN {X 0,Y 255.203,Z 612.621,A -85,B 0,C 180,E1 -20402.554,E2 -20402.554} C_VEL
LIN {X 0,Y 255.479,Z 615.692,A -85,B 0,C 180,E1 -20403.053,E2 -20403.053} C_VEL
LIN {X 0,Y 251.619,Z 630.187,A -85,B 0,C 180,E1 -20404.788,E2 -20404.788} C_VEL
LIN {X 0,Y 247.494,Z 643.862,A -85,B 0,C 180,E1 -20406.795,E2 -20406.795} C_VEL
LIN {X 0,Y 243.518,Z 655.607,A -85,B 0,C 180,E1 -20408.852,E2 -20408.852} C_VEL
LIN {X 0,Y 239.01,Z 668.265,A -85,B 0,C 180,E1 -20411.571,E2 -20411.571} C_VEL
LIN {X 0,Y 234.9,Z 678.967,A -85,B 0,C 180,E1 -20414.377,E2 -20414.377} C_VEL
LIN {X 0,Y 231.19,Z 688.174,A -85,B 0,C 180,E1 -20417.266,E2 -20417.266} C_VEL
LIN {X 0,Y 227.805,Z 696.915,A -85,B 0,C 180,E1 -20420.587,E2 -20420.587} C_VEL
LIN {X 0,Y 224.449,Z 705.442,A -85,B 0,C 180,E1 -20424.608,E2 -20424.608} C_VEL
LIN {X 0,Y 222.25,Z 711.442,A -85,B 0,C 180,E1 -20428.186,E2 -20428.186} C_VEL
LIN {X 0,Y 220.647,Z 716.309,A -85,B 0,C 180,E1 -20431.823,E2 -20431.823} C_VEL
LIN {X 0,Y 219.607,Z 720.145,A -85,B 0,C 180,E1 -20435.507,E2 -20435.507} C_VEL
LIN {X 0,Y 218.916,Z 722.9,A -85,B 0,C 180,E1 -20439.235,E2 -20439.235} C_VEL
LIN {X 0,Y 218.631,Z 724.75,A -85,B 0,C 180,E1 -20443.002,E2 -20443.002} C_VEL
LIN {X 0,Y 218.642,Z 725.547,A -85,B 0,C 180,E1 -20446.813,E2 -20446.813} C_VEL
LIN {X 0,Y 219.027,Z 725.413,A -85,B 0,C 180,E1 -20450.666,E2 -20450.666} C_VEL
LIN {X 0,Y 219.85,Z 724.237,A -85,B 0,C 180,E1 -20454.553,E2 -20454.553} C_VEL
LIN {X 0,Y 221.314,Z 721.988,A -85,B 0,C 180,E1 -20458.444,E2 -20458.444} C_VEL
LIN {X 0,Y 223.424,Z 718.678,A -85,B 0,C 180,E1 -20462.324,E2 -20462.324} C_VEL
LIN {X 0,Y 226.226,Z 714.085,A -85,B 0,C 180,E1 -20466.172,E2 -20466.172} C_VEL
LIN {X 0,Y 229.885,Z 708.216,A -85,B 0,C 180,E1 -20469.939,E2 -20469.939} C_VEL
LIN {X 0,Y 234.421,Z 700.93,A -85,B 0,C 180,E1 -20473.591,E2 -20473.591} C_VEL
LIN {X 0,Y 239.803,Z 692.01,A -85,B 0,C 180,E1 -20477.109,E2 -20477.109} C_VEL
LIN {X 0,Y 245.111,Z 682.641,A -85,B 0,C 180,E1 -20480.081,E2 -20480.081} C_VEL
LIN {X 0,Y 250.179,Z 673.186,A -85,B 0,C 180,E1 -20482.519,E2 -20482.519} C_VEL
LIN {X 0,Y 256.06,Z 661.33,A -85,B 0,C 180,E1 -20485.047,E2 -20485.047} C_VEL
LIN {X 0,Y 261.735,Z 648.737,A -85,B 0,C 180,E1 -20487.23,E2 -20487.23} C_VEL
LIN {X 0,Y 266.583,Z 636.61,A -85,B 0,C 180,E1 -20488.956,E2 -20488.956} C_VEL
LIN {X 0,Y 270.055,Z 626.927,A -85,B 0,C 180,E1 -20490.14,E2 -20490.14} C_VEL
LIN {X 0,Y 270.263,Z 625.372,A -85,B 0,C 180,E1 -20490.39,E2 -20490.39} C_VEL
LIN {X 0,Y 268.957,Z 615.626,A -85,B 0,C 180,E1 -20492.673,E2 -20492.673} C_VEL
LIN {X 0,Y 267.082,Z 607.845,A -85,B 0,C 180,E1 -20494.684,E2 -20494.684} C_VEL
LIN {X 0,Y 264.207,Z 599.998,A -85,B 0,C 180,E1 -20497.034,E2 -20497.034} C_VEL
LIN {X 0,Y 260.964,Z 592.557,A -85,B 0,C 180,E1 -20499.506,E2 -20499.506} C_VEL
LIN {X 0,Y 256.983,Z 584.958,A -85,B 0,C 180,E1 -20502.441,E2 -20502.441} C_VEL
LIN {X 0,Y 255.136,Z 581.668,A -85,B 0,C 180,E1 -20503.856,E2 -20503.856} C_VEL
LIN {X 0,Y 252.636,Z 577.492,A -85,B 0,C 180,E1 -20505.808,E2 -20505.808} C_VEL
LIN {X 0,Y 249.952,Z 573.179,A -85,B 0,C 180,E1 -20508.084,E2 -20508.084} C_VEL
LIN {X 0,Y 247.251,Z 569.444,A -85,B 0,C 180,E1 -20510.489,E2 -20510.489} C_VEL
LIN {X 0,Y 246.357,Z 568.089,A -85,B 0,C 180,E1 -20511.386,E2 -20511.386} C_VEL
LIN {X 0,Y 243.374,Z 564.121,A -85,B 0,C 180,E1 -20514.718,E2 -20514.718} C_VEL
LIN {X 0,Y 242.813,Z 563.297,A -85,B 0,C 180,E1 -20515.434,E2 -20515.434} C_VEL
LIN {X 0,Y 239.096,Z 558.659,A -85,B 0,C 180,E1 -20522.063,E2 -20522.063} C_VEL
LIN {X 0,Y 238.049,Z 558.597,A -85,B 0,C 180,E1 -20528.488,E2 -20528.488} C_VEL
LIN {X 0,Y 239.341,Z 560.339,A -85,B 0,C 180,E1 -20533.856,E2 -20533.856} C_VEL
LIN {X 0,Y 240.411,Z 561.673,A -85,B 0,C 180,E1 -20536.018,E2 -20536.018} C_VEL
LIN {X 0,Y 246.327,Z 569.299,A -85,B 0,C 180,E1 -20543.319,E2 -20543.319} C_VEL
LIN {X 0,Y 250.066,Z 575.126,A -85,B 0,C 180,E1 -20546.585,E2 -20546.585} C_VEL
LIN {X 0,Y 253.863,Z 582.927,A -85,B 0,C 180,E1 -20549.659,E2 -20549.659} C_VEL
LIN {X 0,Y 254.807,Z 584.881,A -85,B 0,C 180,E1 -20550.368,E2 -20550.368} C_VEL
LIN {X 0,Y 255.75,Z 586.912,A -85,B 0,C 180,E1 -20551.086,E2 -20551.086} C_VEL
LIN {X 0,Y 256.682,Z 590.955,A -85,B 0,C 180,E1 -20552.023,E2 -20552.023} C_VEL
LIN {X 0,Y 257.83,Z 605.245,A -85,B 0,C 180,E1 -20554.493,E2 -20554.493} C_VEL
LIN {X 0,Y 258.37,Z 608.018,A -85,B 0,C 180,E1 -20555.133,E2 -20555.133} C_VEL
LIN {X 0,Y 259.934,Z 613.276,A -85,B 0,C 180,E1 -20556.5,E2 -20556.5} C_VEL
LIN {X 0,Y 260.661,Z 617.149,A -85,B 0,C 180,E1 -20557.386,E2 -20557.386} C_VEL
LIN {X 0,Y 260.768,Z 629.988,A -85,B 0,C 180,E1 -20559.585,E2 -20559.585} C_VEL
LIN {X 0,Y 260.08,Z 641.209,A -85,B 0,C 180,E1 -20561.483,E2 -20561.483} C_VEL
LIN {X 0,Y 258.021,Z 656.063,A -85,B 0,C 180,E1 -20564.015,E2 -20564.015} C_VEL
LIN {X 0,Y 257.449,Z 659.071,A -85,B 0,C 180,E1 -20564.563,E2 -20564.563} C_VEL
LIN {X 0,Y 252.07,Z 671.732,A -85,B 0,C 180,E1 -20566.308,E2 -20566.308} C_VEL
LIN {X 0,Y 246.287,Z 684.121,A -85,B 0,C 180,E1 -20568.439,E2 -20568.439} C_VEL
LIN {X 0,Y 240.085,Z 696.278,A -85,B 0,C 180,E1 -20570.999,E2 -20570.999} C_VEL
LIN {X 0,Y 233.753,Z 708.055,A -85,B 0,C 180,E1 -20574.109,E2 -20574.109} C_VEL
LIN {X 0,Y 228.189,Z 717.998,A -85,B 0,C 180,E1 -20577.388,E2 -20577.388} C_VEL
LIN {X 0,Y 223.392,Z 726.436,A -85,B 0,C 180,E1 -20580.817,E2 -20580.817} C_VEL
LIN {X 0,Y 219.461,Z 733.433,A -85,B 0,C 180,E1 -20584.387,E2 -20584.387} C_VEL
LIN {X 0,Y 216.395,Z 739.273,A -85,B 0,C 180,E1 -20588.071,E2 -20588.071} C_VEL
LIN {X 0,Y 213.953,Z 744.517,A -85,B 0,C 180,E1 -20592.286,E2 -20592.286} C_VEL
LIN {X 0,Y 212.383,Z 748.427,A -85,B 0,C 180,E1 -20596.609,E2 -20596.609} C_VEL
LIN {X 0,Y 211.744,Z 750.857,A -85,B 0,C 180,E1 -20600.449,E2 -20600.449} C_VEL
LIN {X 0,Y 211.847,Z 752.345,A -85,B 0,C 180,E1 -20604.402,E2 -20604.402} C_VEL
LIN {X 0,Y 211.872,Z 752.773,A -85,B 0,C 180,E1 -20608.101,E2 -20608.101} C_VEL
LIN {X 0,Y 211.974,Z 752.657,A -85,B 0,C 180,E1 -20610.002,E2 -20610.002} C_VEL
LIN {X 0,Y 211.888,Z 751.529,A -85,B 0,C 180,E1 -20613.806,E2 -20613.806} C_VEL
LIN {X 0,Y 211.907,Z 750.582,A -85,B 0,C 180,E1 -20615.76,E2 -20615.76} C_VEL
LIN {X 0,Y 211.844,Z 747.935,A -85,B 0,C 180,E1 -20619.55,E2 -20619.55} C_VEL
LIN {X 0,Y 212.459,Z 744.151,A -85,B 0,C 180,E1 -20623.391,E2 -20623.391} C_VEL
LIN {X 0,Y 213.775,Z 738.76,A -85,B 0,C 180,E1 -20627.564,E2 -20627.564} C_VEL
LIN {X 0,Y 215.556,Z 733.109,A -85,B 0,C 180,E1 -20631.019,E2 -20631.019} C_VEL
LIN {X 0,Y 220.242,Z 725.537,A -85,B 0,C 180,E1 -20636.687,E2 -20636.687} C_VEL
LIN {X 0,Y 225.525,Z 718.34,A -85,B 0,C 180,E1 -20640.945,E2 -20640.945} C_VEL
LIN {X 0,Y 233.949,Z 708.177,A -85,B 0,C 180,E1 -20645.798,E2 -20645.798} C_VEL
LIN {X 0,Y 244.573,Z 696.38,A -85,B 0,C 180,E1 -20650.284,E2 -20650.284} C_VEL
LIN {X 0,Y 257.231,Z 683.345,A -85,B 0,C 180,E1 -20654.165,E2 -20654.165} C_VEL
LIN {X 0,Y 271.202,Z 669.59,A -85,B 0,C 180,E1 -20657.362,E2 -20657.362} C_VEL
LIN {X 0,Y 272.562,Z 668.183,A -85,B 0,C 180,E1 -20657.722,E2 -20657.722} C_VEL
LIN {X 0,Y 273.093,Z 667.543,A -85,B 0,C 180,E1 -20658.003,E2 -20658.003} C_VEL
LIN {X 0,Y 261.72,Z 675.863,A -85,B 0,C 180,E1 -20660.873,E2 -20660.873} C_VEL
LIN {X 0,Y 250.21,Z 684.018,A -85,B 0,C 180,E1 -20664.546,E2 -20664.546} C_VEL
LIN {X 0,Y 240.818,Z 690.453,A -85,B 0,C 180,E1 -20668.312,E2 -20668.312} C_VEL
LIN {X 0,Y 234.706,Z 694.501,A -85,B 0,C 180,E1 -20671.374,E2 -20671.374} C_VEL
LIN {X 0,Y 226.993,Z 699.151,A -85,B 0,C 180,E1 -20676.266,E2 -20676.266} C_VEL
LIN {X 0,Y 222.908,Z 701.349,A -85,B 0,C 180,E1 -20679.708,E2 -20679.708} C_VEL
LIN {X 0,Y 219.564,Z 702.799,A -85,B 0,C 180,E1 -20683.258,E2 -20683.258} C_VEL
LIN {X 0,Y 217.025,Z 703.422,A -85,B 0,C 180,E1 -20686.899,E2 -20686.899} C_VEL
LIN {X 0,Y 215.302,Z 703.255,A -85,B 0,C 180,E1 -20690.607,E2 -20690.607} C_VEL
LIN {X 0,Y 213.896,Z 702.249,A -85,B 0,C 180,E1 -20694.344,E2 -20694.344} C_VEL
LIN {X 0,Y 213.035,Z 700.39,A -85,B 0,C 180,E1 -20698.11,E2 -20698.11} C_VEL
LIN {X 0,Y 212.866,Z 697.55,A -85,B 0,C 180,E1 -20701.893,E2 -20701.893} C_VEL
LIN {X 0,Y 213.015,Z 695.774,A -85,B 0,C 180,E1 -20703.784,E2 -20703.784} C_VEL
LIN {X 0,Y 213.175,Z 691.549,A -85,B 0,C 180,E1 -20707.579,E2 -20707.579} C_VEL
LIN {X 0,Y 213.834,Z 686.143,A -85,B 0,C 180,E1 -20711.374,E2 -20711.374} C_VEL
LIN {X 0,Y 214.917,Z 679.577,A -85,B 0,C 180,E1 -20715.166,E2 -20715.166} C_VEL
LIN {X 0,Y 216.709,Z 671.742,A -85,B 0,C 180,E1 -20718.924,E2 -20718.924} C_VEL
LIN {X 0,Y 219.109,Z 662.41,A -85,B 0,C 180,E1 -20722.639,E2 -20722.639} C_VEL
LIN {X 0,Y 222.2,Z 651.357,A -85,B 0,C 180,E1 -20726.284,E2 -20726.284} C_VEL
LIN {X 0,Y 225.45,Z 639.54,A -85,B 0,C 180,E1 -20729.552,E2 -20729.552} C_VEL
LIN {X 0,Y 229.092,Z 626.924,A -85,B 0,C 180,E1 -20732.471,E2 -20732.471} C_VEL
LIN {X 0,Y 232.739,Z 613.919,A -85,B 0,C 180,E1 -20735.012,E2 -20735.012} C_VEL
LIN {X 0,Y 236.732,Z 598.821,A -85,B 0,C 180,E1 -20737.489,E2 -20737.489} C_VEL
LIN {X 0,Y 238.36,Z 591.678,A -85,B 0,C 180,E1 -20738.526,E2 -20738.526} C_VEL
LIN {X 0,Y 233.741,Z 578.259,A -85,B 0,C 180,E1 -20741.261,E2 -20741.261} C_VEL
LIN {X 0,Y 228.826,Z 565.375,A -85,B 0,C 180,E1 -20743.798,E2 -20743.798} C_VEL
LIN {X 0,Y 223.039,Z 551.888,A -85,B 0,C 180,E1 -20746.448,E2 -20746.448} C_VEL
LIN {X 0,Y 220.859,Z 547.973,A -85,B 0,C 180,E1 -20747.273,E2 -20747.273} C_VEL
LIN {X 0,Y 221.925,Z 548.69,A -85,B 0,C 180,E1 -20747.74,E2 -20747.74} C_VEL
LIN {X 0,Y 223.634,Z 550.892,A -85,B 0,C 180,E1 -20748.419,E2 -20748.419} C_VEL
LIN {X 0,Y 227.515,Z 556.952,A -85,B 0,C 180,E1 -20750.002,E2 -20750.002} C_VEL
LIN {X 0,Y 230.097,Z 560.967,A -85,B 0,C 180,E1 -20751.034,E2 -20751.034} C_VEL
LIN {X 0,Y 235.958,Z 571.334,A -85,B 0,C 180,E1 -20753.475,E2 -20753.475} C_VEL
LIN {X 0,Y 241.543,Z 583.511,A -85,B 0,C 180,E1 -20756.024,E2 -20756.024} C_VEL
LIN {X 0,Y 244.839,Z 593.645,A -85,B 0,C 180,E1 -20757.924,E2 -20757.924} C_VEL
LIN {X 0,Y 247.634,Z 605.793,A -85,B 0,C 180,E1 -20760.113,E2 -20760.113} C_VEL
LIN {X 0,Y 249.525,Z 616.31,A -85,B 0,C 180,E1 -20762.043,E2 -20762.043} C_VEL
LIN {X 0,Y 249.33,Z 618.366,A -85,B 0,C 180,E1 -20762.333,E2 -20762.333} C_VEL
LIN {X 0,Y 245.325,Z 632.541,A -85,B 0,C 180,E1 -20764.094,E2 -20764.094} C_VEL
LIN {X 0,Y 241.076,Z 645.887,A -85,B 0,C 180,E1 -20766.139,E2 -20766.139} C_VEL
LIN {X 0,Y 236.995,Z 657.369,A -85,B 0,C 180,E1 -20768.241,E2 -20768.241} C_VEL
LIN {X 0,Y 232.35,Z 669.831,A -85,B 0,C 180,E1 -20771.023,E2 -20771.023} C_VEL
LIN {X 0,Y 228.133,Z 680.425,A -85,B 0,C 180,E1 -20773.902,E2 -20773.902} C_VEL
LIN {X 0,Y 223.839,Z 690.668,A -85,B 0,C 180,E1 -20777.302,E2 -20777.302} C_VEL
LIN {X 0,Y 220.332,Z 699.247,A -85,B 0,C 180,E1 -20780.821,E2 -20780.821} C_VEL
LIN {X 0,Y 217.402,Z 706.452,A -85,B 0,C 180,E1 -20784.433,E2 -20784.433} C_VEL
LIN {X 0,Y 215.142,Z 712.393,A -85,B 0,C 180,E1 -20788.126,E2 -20788.126} C_VEL
LIN {X 0,Y 213.544,Z 717.133,A -85,B 0,C 180,E1 -20791.884,E2 -20791.884} C_VEL
LIN {X 0,Y 212.495,Z 720.885,A -85,B 0,C 180,E1 -20795.692,E2 -20795.692} C_VEL
LIN {X 0,Y 211.779,Z 723.559,A -85,B 0,C 180,E1 -20799.549,E2 -20799.549} C_VEL
LIN {X 0,Y 211.542,Z 725.295,A -85,B 0,C 180,E1 -20803.446,E2 -20803.446} C_VEL
LIN {X 0,Y 211.584,Z 726.042,A -85,B 0,C 180,E1 -20807.392,E2 -20807.392} C_VEL
LIN {X 0,Y 212.169,Z 725.671,A -85,B 0,C 180,E1 -20811.951,E2 -20811.951} C_VEL
LIN {X 0,Y 213.012,Z 724.564,A -85,B 0,C 180,E1 -20815.396,E2 -20815.396} C_VEL
LIN {X 0,Y 214.645,Z 722.197,A -85,B 0,C 180,E1 -20819.413,E2 -20819.413} C_VEL
LIN {X 0,Y 216.959,Z 718.762,A -85,B 0,C 180,E1 -20823.411,E2 -20823.411} C_VEL
LIN {X 0,Y 220.077,Z 714.101,A -85,B 0,C 180,E1 -20827.352,E2 -20827.352} C_VEL
LIN {X 0,Y 224.035,Z 708.092,A -85,B 0,C 180,E1 -20831.203,E2 -20831.203} C_VEL
LIN {X 0,Y 228.912,Z 700.662,A -85,B 0,C 180,E1 -20834.918,E2 -20834.918} C_VEL
LIN {X 0,Y 233.883,Z 692.857,A -85,B 0,C 180,E1 -20838.046,E2 -20838.046} C_VEL
LIN {X 0,Y 239.406,Z 683.527,A -85,B 0,C 180,E1 -20841.068,E2 -20841.068} C_VEL
LIN {X 0,Y 244.677,Z 674.16,A -85,B 0,C 180,E1 -20843.535,E2 -20843.535} C_VEL
LIN {X 0,Y 250.712,Z 662.519,A -85,B 0,C 180,E1 -20846.068,E2 -20846.068} C_VEL
LIN {X 0,Y 256.367,Z 650.567,A -85,B 0,C 180,E1 -20848.189,E2 -20848.189} C_VEL
LIN {X 0,Y 261.641,Z 637.919,A -85,B 0,C 180,E1 -20850.024,E2 -20850.024} C_VEL
LIN {X 0,Y 264.89,Z 629.254,A -85,B 0,C 180,E1 -20851.105,E2 -20851.105} C_VEL
LIN {X 0,Y 264.861,Z 625.925,A -85,B 0,C 180,E1 -20851.842,E2 -20851.842} C_VEL
LIN {X 0,Y 263.769,Z 617.586,A -85,B 0,C 180,E1 -20853.919,E2 -20853.919} C_VEL
LIN {X 0,Y 262.116,Z 610.844,A -85,B 0,C 180,E1 -20855.822,E2 -20855.822} C_VEL
LIN {X 0,Y 258.681,Z 601.345,A -85,B 0,C 180,E1 -20858.9,E2 -20858.9} C_VEL
LIN {X 0,Y 255.502,Z 594.218,A -85,B 0,C 180,E1 -20861.558,E2 -20861.558} C_VEL
LIN {X 0,Y 252.839,Z 588.66,A -85,B 0,C 180,E1 -20863.861,E2 -20863.861} C_VEL
LIN {X 0,Y 250.527,Z 584.617,A -85,B 0,C 180,E1 -20865.79,E2 -20865.79} C_VEL
LIN {X 0,Y 247.433,Z 579.468,A -85,B 0,C 180,E1 -20868.635,E2 -20868.635} C_VEL
LIN {X 0,Y 244.881,Z 575.449,A -85,B 0,C 180,E1 -20871.229,E2 -20871.229} C_VEL
LIN {X 0,Y 241.14,Z 570.095,A -85,B 0,C 180,E1 -20875.821,E2 -20875.821} C_VEL
LIN {X 0,Y 237.988,Z 565.721,A -85,B 0,C 180,E1 -20882.072,E2 -20882.072} C_VEL
LIN {X 0,Y 236.974,Z 565.449,A -85,B 0,C 180,E1 -20886.812,E2 -20886.812} C_VEL
LIN {X 0,Y 237.587,Z 566.577,A -85,B 0,C 180,E1 -20891.95,E2 -20891.95} C_VEL
LIN {X 0,Y 239.066,Z 568.385,A -85,B 0,C 180,E1 -20895.56,E2 -20895.56} C_VEL
LIN {X 0,Y 244.59,Z 575.977,A -85,B 0,C 180,E1 -20902.913,E2 -20902.913} C_VEL
LIN {X 0,Y 247.827,Z 581.424,A -85,B 0,C 180,E1 -20906.018,E2 -20906.018} C_VEL
LIN {X 0,Y 251.066,Z 588.752,A -85,B 0,C 180,E1 -20908.987,E2 -20908.987} C_VEL
LIN {X 0,Y 253.221,Z 593.799,A -85,B 0,C 180,E1 -20910.788,E2 -20910.788} C_VEL
LIN {X 0,Y 257.668,Z 605.495,A -85,B 0,C 180,E1 -20914.468,E2 -20914.468} C_VEL
LIN {X 0,Y 258.37,Z 608.018,A -85,B 0,C 180,E1 -20915.133,E2 -20915.133} C_VEL
LIN {X 0,Y 258.891,Z 610.78,A -85,B 0,C 180,E1 -20915.744,E2 -20915.744} C_VEL
LIN {X 0,Y 258.918,Z 615.598,A -85,B 0,C 180,E1 -20916.51,E2 -20916.51} C_VEL
LIN {X 0,Y 258.275,Z 620.794,A -85,B 0,C 180,E1 -20917.151,E2 -20917.151} C_VEL
LIN {X 0,Y 256.322,Z 631.448,A -85,B 0,C 180,E1 -20918.43,E2 -20918.43} C_VEL
LIN {X 0,Y 255.902,Z 634.755,A -85,B 0,C 180,E1 -20918.952,E2 -20918.952} C_VEL
LIN {X 0,Y 254.934,Z 644.582,A -85,B 0,C 180,E1 -20920.672,E2 -20920.672} C_VEL
LIN {X 0,Y 252.521,Z 658.841,A -85,B 0,C 180,E1 -20923.214,E2 -20923.214} C_VEL
LIN {X 0,Y 252.123,Z 660.695,A -85,B 0,C 180,E1 -20923.555,E2 -20923.555} C_VEL
LIN {X 0,Y 245.769,Z 674.674,A -85,B 0,C 180,E1 -20925.581,E2 -20925.581} C_VEL
LIN {X 0,Y 240.039,Z 686.28,A -85,B 0,C 180,E1 -20927.672,E2 -20927.672} C_VEL
LIN {X 0,Y 233.7,Z 698.075,A -85,B 0,C 180,E1 -20930.282,E2 -20930.282} C_VEL
LIN {X 0,Y 227.832,Z 708.396,A -85,B 0,C 180,E1 -20933.135,E2 -20933.135} C_VEL
LIN {X 0,Y 222.194,Z 717.976,A -85,B 0,C 180,E1 -20936.394,E2 -20936.394} C_VEL
LIN {X 0,Y 217.114,Z 726.323,A -85,B 0,C 180,E1 -20939.888,E2 -20939.888} C_VEL
LIN {X 0,Y 212.972,Z 733.273,A -85,B 0,C 180,E1 -20943.548,E2 -20943.548} C_VEL
LIN {X 0,Y 209.705,Z 739.042,A -85,B 0,C 180,E1 -20947.333,E2 -20947.333} C_VEL
LIN {X 0,Y 206.942,Z 744.507,A -85,B 0,C 180,E1 -20951.971,E2 -20951.971} C_VEL
LIN {X 0,Y 205.386,Z 748.099,A -85,B 0,C 180,E1 -20956.144,E2 -20956.144} C_VEL
LIN {X 0,Y 204.667,Z 750.469,A -85,B 0,C 180,E1 -20960.116,E2 -20960.116} C_VEL
LIN {X 0,Y 204.748,Z 752.016,A -85,B 0,C 180,E1 -20964.512,E2 -20964.512} C_VEL
LIN {X 0,Y 204.8,Z 752.307,A -85,B 0,C 180,E1 -20968.036,E2 -20968.036} C_VEL
LIN {X 0,Y 204.897,Z 752.175,A -85,B 0,C 180,E1 -20970.002,E2 -20970.002} C_VEL
LIN {X 0,Y 204.807,Z 751.007,A -85,B 0,C 180,E1 -20973.937,E2 -20973.937} C_VEL
LIN {X 0,Y 204.814,Z 750.058,A -85,B 0,C 180,E1 -20975.911,E2 -20975.911} C_VEL
LIN {X 0,Y 204.789,Z 747.353,A -85,B 0,C 180,E1 -20979.882,E2 -20979.882} C_VEL
LIN {X 0,Y 205.48,Z 743.507,A -85,B 0,C 180,E1 -20983.854,E2 -20983.854} C_VEL
LIN {X 0,Y 206.808,Z 738.426,A -85,B 0,C 180,E1 -20987.915,E2 -20987.915} C_VEL
LIN {X 0,Y 208.822,Z 732.74,A -85,B 0,C 180,E1 -20991.73,E2 -20991.73} C_VEL
LIN {X 0,Y 213.566,Z 725.896,A -85,B 0,C 180,E1 -20997.315,E2 -20997.315} C_VEL
LIN {X 0,Y 219.418,Z 718.73,A -85,B 0,C 180,E1 -21001.906,E2 -21001.906} C_VEL
LIN {X 0,Y 228.19,Z 709.176,A -85,B 0,C 180,E1 -21006.797,E2 -21006.797} C_VEL
LIN {X 0,Y 239.341,Z 697.933,A -85,B 0,C 180,E1 -21011.354,E2 -21011.354} C_VEL
LIN {X 0,Y 253.602,Z 684.528,A -85,B 0,C 180,E1 -21015.531,E2 -21015.531} C_VEL
LIN {X 0,Y 264.781,Z 674.407,A -85,B 0,C 180,E1 -21018.006,E2 -21018.006} C_VEL
LIN {X 0,Y 252.602,Z 682.328,A -85,B 0,C 180,E1 -21021.245,E2 -21021.245} C_VEL
LIN {X 0,Y 240.564,Z 689.877,A -85,B 0,C 180,E1 -21025.273,E2 -21025.273} C_VEL
LIN {X 0,Y 231.91,Z 695.007,A -85,B 0,C 180,E1 -21028.991,E2 -21028.991} C_VEL
LIN {X 0,Y 223.252,Z 699.776,A -85,B 0,C 180,E1 -21033.851,E2 -21033.851} C_VEL
LIN {X 0,Y 216.462,Z 702.992,A -85,B 0,C 180,E1 -21039.076,E2 -21039.076} C_VEL
LIN {X 0,Y 211.471,Z 704.489,A -85,B 0,C 180,E1 -21044.582,E2 -21044.582} C_VEL
LIN {X 0,Y 209.19,Z 704.5,A -85,B 0,C 180,E1 -21048.372,E2 -21048.372} C_VEL
LIN {X 0,Y 207.561,Z 703.748,A -85,B 0,C 180,E1 -21052.217,E2 -21052.217} C_VEL
LIN {X 0,Y 206.31,Z 702.12,A -85,B 0,C 180,E1 -21056.094,E2 -21056.094} C_VEL
LIN {X 0,Y 205.801,Z 699.619,A -85,B 0,C 180,E1 -21060.001,E2 -21060.001} C_VEL
LIN {X 0,Y 205.925,Z 696.133,A -85,B 0,C 180,E1 -21063.915,E2 -21063.915} C_VEL
LIN {X 0,Y 206.113,Z 691.676,A -85,B 0,C 180,E1 -21067.84,E2 -21067.84} C_VEL
LIN {X 0,Y 206.817,Z 686.19,A -85,B 0,C 180,E1 -21071.765,E2 -21071.765} C_VEL
LIN {X 0,Y 207.99,Z 679.389,A -85,B 0,C 180,E1 -21075.684,E2 -21075.684} C_VEL
LIN {X 0,Y 209.924,Z 671.309,A -85,B 0,C 180,E1 -21079.561,E2 -21079.561} C_VEL
LIN {X 0,Y 212.452,Z 661.751,A -85,B 0,C 180,E1 -21083.39,E2 -21083.39} C_VEL
LIN {X 0,Y 215.716,Z 650.504,A -85,B 0,C 180,E1 -21087.138,E2 -21087.138} C_VEL
LIN {X 0,Y 219.084,Z 638.701,A -85,B 0,C 180,E1 -21090.425,E2 -21090.425} C_VEL
LIN {X 0,Y 223.276,Z 624.487,A -85,B 0,C 180,E1 -21093.696,E2 -21093.696} C_VEL
LIN {X 0,Y 227.254,Z 610.509,A -85,B 0,C 180,E1 -21096.376,E2 -21096.376} C_VEL
LIN {X 0,Y 231.291,Z 595.256,A -85,B 0,C 180,E1 -21098.809,E2 -21098.809} C_VEL
LIN {X 0,Y 231.646,Z 593.789,A -85,B 0,C 180,E1 -21099.017,E2 -21099.017} C_VEL
LIN {X 0,Y 227.361,Z 580.852,A -85,B 0,C 180,E1 -21101.754,E2 -21101.754} C_VEL
LIN {X 0,Y 222.576,Z 568.039,A -85,B 0,C 180,E1 -21104.404,E2 -21104.404} C_VEL
LIN {X 0,Y 217.656,Z 556.451,A -85,B 0,C 180,E1 -21106.793,E2 -21106.793} C_VEL
LIN {X 0,Y 218.386,Z 556.762,A -85,B 0,C 180,E1 -21107.066,E2 -21107.066} C_VEL
LIN {X 0,Y 220.304,Z 556.546,A -85,B 0,C 180,E1 -21107.699,E2 -21107.699} C_VEL
LIN {X 0,Y 226.268,Z 566.238,A -85,B 0,C 180,E1 -21110.33,E2 -21110.33} C_VEL
LIN {X 0,Y 231.841,Z 576.644,A -85,B 0,C 180,E1 -21112.868,E2 -21112.868} C_VEL
LIN {X 0,Y 236.828,Z 588.289,A -85,B 0,C 180,E1 -21115.439,E2 -21115.439} C_VEL
LIN {X 0,Y 239.497,Z 597.035,A -85,B 0,C 180,E1 -21117.163,E2 -21117.163} C_VEL
LIN {X 0,Y 242.126,Z 609.372,A -85,B 0,C 180,E1 -21119.477,E2 -21119.477} C_VEL
LIN {X 0,Y 243.702,Z 619.039,A -85,B 0,C 180,E1 -21121.348,E2 -21121.348} C_VEL
LIN {X 0,Y 239.456,Z 633.521,A -85,B 0,C 180,E1 -21123.174,E2 -21123.174} C_VEL
LIN {X 0,Y 235.089,Z 646.772,A -85,B 0,C 180,E1 -21125.257,E2 -21125.257} C_VEL
LIN {X 0,Y 230.5,Z 659.132,A -85,B 0,C 180,E1 -21127.595,E2 -21127.595} C_VEL
LIN {X 0,Y 225.714,Z 671.38,A -85,B 0,C 180,E1 -21130.443,E2 -21130.443} C_VEL
LIN {X 0,Y 221.383,Z 681.843,A -85,B 0,C 180,E1 -21133.397,E2 -21133.397} C_VEL
LIN {X 0,Y 216.966,Z 691.955,A -85,B 0,C 180,E1 -21136.893,E2 -21136.893} C_VEL
LIN {X 0,Y 213.372,Z 700.381,A -85,B 0,C 180,E1 -21140.519,E2 -21140.519} C_VEL
LIN {X 0,Y 210.361,Z 707.45,A -85,B 0,C 180,E1 -21144.246,E2 -21144.246} C_VEL
LIN {X 0,Y 208.037,Z 713.318,A -85,B 0,C 180,E1 -21148.062,E2 -21148.062} C_VEL
LIN {X 0,Y 206.425,Z 717.952,A -85,B 0,C 180,E1 -21151.949,E2 -21151.949} C_VEL
LIN {X 0,Y 205.184,Z 722.13,A -85,B 0,C 180,E1 -21156.621,E2 -21156.621} C_VEL
LIN {X 0,Y 204.664,Z 724.211,A -85,B 0,C 180,E1 -21159.884,E2 -21159.884} C_VEL
LIN {X 0,Y 204.433,Z 725.841,A -85,B 0,C 180,E1 -21163.922,E2 -21163.922} C_VEL
LIN {X 0,Y 204.543,Z 726.536,A -85,B 0,C 180,E1 -21168.011,E2 -21168.011} C_VEL
LIN {X 0,Y 205.169,Z 726.133,A -85,B 0,C 180,E1 -21172.348,E2 -21172.348} C_VEL
LIN {X 0,Y 206.227,Z 724.865,A -85,B 0,C 180,E1 -21176.294,E2 -21176.294} C_VEL
LIN {X 0,Y 208.039,Z 722.406,A -85,B 0,C 180,E1 -21180.444,E2 -21180.444} C_VEL
LIN {X 0,Y 210.604,Z 718.844,A -85,B 0,C 180,E1 -21184.559,E2 -21184.559} C_VEL
LIN {X 0,Y 214.021,Z 714.111,A -85,B 0,C 180,E1 -21188.6,E2 -21188.6} C_VEL
LIN {X 0,Y 218.32,Z 707.982,A -85,B 0,C 180,E1 -21192.53,E2 -21192.53} C_VEL
LIN {X 0,Y 223.559,Z 700.403,A -85,B 0,C 180,E1 -21196.303,E2 -21196.303} C_VEL
LIN {X 0,Y 229.622,Z 691.159,A -85,B 0,C 180,E1 -21199.919,E2 -21199.919} C_VEL
LIN {X 0,Y 235.561,Z 681.477,A -85,B 0,C 180,E1 -21202.944,E2 -21202.944} C_VEL
LIN {X 0,Y 241.163,Z 671.768,A -85,B 0,C 180,E1 -21205.409,E2 -21205.409} C_VEL
LIN {X 0,Y 247.21,Z 660.185,A -85,B 0,C 180,E1 -21207.82,E2 -21207.82} C_VEL
LIN {X 0,Y 252.908,Z 648.264,A -85,B 0,C 180,E1 -21209.84,E2 -21209.84} C_VEL
LIN {X 0,Y 258.697,Z 634.582,A -85,B 0,C 180,E1 -21211.735,E2 -21211.735} C_VEL
LIN {X 0,Y 259.865,Z 631.143,A -85,B 0,C 180,E1 -21212.19,E2 -21212.19} C_VEL
LIN {X 0,Y 259.187,Z 623.003,A -85,B 0,C 180,E1 -21214.287,E2 -21214.287} C_VEL
LIN {X 0,Y 257.802,Z 616.075,A -85,B 0,C 180,E1 -21216.29,E2 -21216.29} C_VEL
LIN {X 0,Y 255.206,Z 607.919,A -85,B 0,C 180,E1 -21219.022,E2 -21219.022} C_VEL
LIN {X 0,Y 252.783,Z 601.687,A -85,B 0,C 180,E1 -21221.353,E2 -21221.353} C_VEL
LIN {X 0,Y 249.488,Z 594.407,A -85,B 0,C 180,E1 -21224.477,E2 -21224.477} C_VEL
LIN {X 0,Y 245.014,Z 586.008,A -85,B 0,C 180,E1 -21228.94,E2 -21228.94} C_VEL
LIN {X 0,Y 242.802,Z 582.256,A -85,B 0,C 180,E1 -21231.468,E2 -21231.468} C_VEL
LIN {X 0,Y 241.574,Z 580.535,A -85,B 0,C 180,E1 -21232.897,E2 -21232.897} C_VEL
LIN {X 0,Y 239.451,Z 576.931,A -85,B 0,C 180,E1 -21235.997,E2 -21235.997} C_VEL
LIN {X 0,Y 236.481,Z 572.563,A -85,B 0,C 180,E1 -21242.554,E2 -21242.554} C_VEL
LIN {X 0,Y 235.731,Z 572.636,A -85,B 0,C 180,E1 -21248.572,E2 -21248.572} C_VEL
LIN {X 0,Y 236.931,Z 574.327,A -85,B 0,C 180,E1 -21253.727,E2 -21253.727} C_VEL
LIN {X 0,Y 237.671,Z 575.393,A -85,B 0,C 180,E1 -21255.433,E2 -21255.433} C_VEL
LIN {X 0,Y 242.648,Z 582.539,A -85,B 0,C 180,E1 -21262.477,E2 -21262.477} C_VEL
LIN {X 0,Y 245.338,Z 587.522,A -85,B 0,C 180,E1 -21265.391,E2 -21265.391} C_VEL
LIN {X 0,Y 248.185,Z 594.527,A -85,B 0,C 180,E1 -21268.314,E2 -21268.314} C_VEL
LIN {X 0,Y 250.127,Z 599.678,A -85,B 0,C 180,E1 -21270.206,E2 -21270.206} C_VEL
LIN {X 0,Y 254.069,Z 611.195,A -85,B 0,C 180,E1 -21273.92,E2 -21273.92} C_VEL
LIN {X 0,Y 255.846,Z 618.39,A -85,B 0,C 180,E1 -21275.875,E2 -21275.875} C_VEL
LIN {X 0,Y 256.285,Z 620.844,A -85,B 0,C 180,E1 -21276.452,E2 -21276.452} C_VEL
LIN {X 0,Y 255.921,Z 634.468,A -85,B 0,C 180,E1 -21278.901,E2 -21278.901} C_VEL
LIN {X 0,Y 255.902,Z 634.755,A -85,B 0,C 180,E1 -21278.952,E2 -21278.952} C_VEL
LIN {X 0,Y 255.073,Z 639.724,A -85,B 0,C 180,E1 -21279.68,E2 -21279.68} C_VEL
LIN {X 0,Y 251.995,Z 648.336,A -85,B 0,C 180,E1 -21280.602,E2 -21280.602} C_VEL
LIN {X 0,Y 248.558,Z 656.686,A -85,B 0,C 180,E1 -21281.555,E2 -21281.555} C_VEL
LIN {X 0,Y 247.129,Z 661.287,A -85,B 0,C 180,E1 -21282.314,E2 -21282.314} C_VEL
LIN {X 0,Y 245.686,Z 664.919,A -85,B 0,C 180,E1 -21282.863,E2 -21282.863} C_VEL
LIN {X 0,Y 239.337,Z 677.941,A -85,B 0,C 180,E1 -21284.867,E2 -21284.867} C_VEL
LIN {X 0,Y 232.906,Z 690.078,A -85,B 0,C 180,E1 -21287.242,E2 -21287.242} C_VEL
LIN {X 0,Y 226.521,Z 701.206,A -85,B 0,C 180,E1 -21289.928,E2 -21289.928} C_VEL
LIN {X 0,Y 220.044,Z 711.822,A -85,B 0,C 180,E1 -21293.109,E2 -21293.109} C_VEL
LIN {X 0,Y 214.8,Z 720.192,A -85,B 0,C 180,E1 -21296.208,E2 -21296.208} C_VEL
LIN {X 0,Y 209.752,Z 728.043,A -85,B 0,C 180,E1 -21299.831,E2 -21299.831} C_VEL
LIN {X 0,Y 205.579,Z 734.654,A -85,B 0,C 180,E1 -21303.616,E2 -21303.616} C_VEL
LIN {X 0,Y 202.327,Z 740.09,A -85,B 0,C 180,E1 -21307.539,E2 -21307.539} C_VEL
LIN {X 0,Y 199.963,Z 744.47,A -85,B 0,C 180,E1 -21311.612,E2 -21311.612} C_VEL
LIN {X 0,Y 198.411,Z 747.774,A -85,B 0,C 180,E1 -21315.646,E2 -21315.646} C_VEL
LIN {X 0,Y 197.611,Z 750.084,A -85,B 0,C 180,E1 -21319.759,E2 -21319.759} C_VEL
LIN {X 0,Y 197.659,Z 751.627,A -85,B 0,C 180,E1 -21324.598,E2 -21324.598} C_VEL
LIN {X 0,Y 197.729,Z 751.842,A -85,B 0,C 180,E1 -21327.965,E2 -21327.965} C_VEL
LIN {X 0,Y 197.823,Z 751.682,A -85,B 0,C 180,E1 -21330.002,E2 -21330.002} C_VEL
LIN {X 0,Y 197.73,Z 750.485,A -85,B 0,C 180,E1 -21334.079,E2 -21334.079} C_VEL
LIN {X 0,Y 197.711,Z 749.504,A -85,B 0,C 180,E1 -21336.124,E2 -21336.124} C_VEL
LIN {X 0,Y 197.723,Z 746.765,A -85,B 0,C 180,E1 -21340.239,E2 -21340.239} C_VEL
LIN {X 0,Y 198.488,Z 742.854,A -85,B 0,C 180,E1 -21344.353,E2 -21344.353} C_VEL
LIN {X 0,Y 199.892,Z 737.85,A -85,B 0,C 180,E1 -21348.449,E2 -21348.449} C_VEL
LIN {X 0,Y 201.467,Z 733.399,A -85,B 0,C 180,E1 -21351.489,E2 -21351.489} C_VEL
LIN {X 0,Y 205.308,Z 728.169,A -85,B 0,C 180,E1 -21356.426,E2 -21356.426} C_VEL
LIN {X 0,Y 210.736,Z 721.909,A -85,B 0,C 180,E1 -21361.128,E2 -21361.128} C_VEL
LIN {X 0,Y 219.417,Z 713.12,A -85,B 0,C 180,E1 -21366.341,E2 -21366.341} C_VEL
LIN {X 0,Y 232.136,Z 701.256,A -85,B 0,C 180,E1 -21371.765,E2 -21371.765} C_VEL
LIN {X 0,Y 245.322,Z 689.826,A -85,B 0,C 180,E1 -21375.744,E2 -21375.744} C_VEL
LIN {X 0,Y 255.178,Z 681.622,A -85,B 0,C 180,E1 -21378.042,E2 -21378.042} C_VEL
LIN {X 0,Y 254.528,Z 681.824,A -85,B 0,C 180,E1 -21378.496,E2 -21378.496} C_VEL
LIN {X 0,Y 241.269,Z 689.388,A -85,B 0,C 180,E1 -21382.287,E2 -21382.287} C_VEL
LIN {X 0,Y 229.686,Z 695.658,A -85,B 0,C 180,E1 -21386.581,E2 -21386.581} C_VEL
LIN {X 0,Y 219.966,Z 700.456,A -85,B 0,C 180,E1 -21391.364,E2 -21391.364} C_VEL
LIN {X 0,Y 214.543,Z 702.883,A -85,B 0,C 180,E1 -21394.796,E2 -21394.796} C_VEL
LIN {X 0,Y 208.032,Z 705.159,A -85,B 0,C 180,E1 -21400.256,E2 -21400.256} C_VEL
LIN {X 0,Y 203.402,Z 705.748,A -85,B 0,C 180,E1 -21406.004,E2 -21406.004} C_VEL
LIN {X 0,Y 201.411,Z 705.147,A -85,B 0,C 180,E1 -21409.953,E2 -21409.953} C_VEL
LIN {X 0,Y 199.861,Z 703.798,A -85,B 0,C 180,E1 -21413.945,E2 -21413.945} C_VEL
LIN {X 0,Y 198.917,Z 701.538,A -85,B 0,C 180,E1 -21417.976,E2 -21417.976} C_VEL
LIN {X 0,Y 198.739,Z 698.389,A -85,B 0,C 180,E1 -21422.027,E2 -21422.027} C_VEL
LIN {X 0,Y 198.824,Z 695.382,A -85,B 0,C 180,E1 -21425.071,E2 -21425.071} C_VEL
LIN {X 0,Y 199.242,Z 690.683,A -85,B 0,C 180,E1 -21429,E2 -21429} C_VEL
LIN {X 0,Y 200.083,Z 684.442,A -85,B 0,C 180,E1 -21433.199,E2 -21433.199} C_VEL
LIN {X 0,Y 201.796,Z 676.201,A -85,B 0,C 180,E1 -21437.743,E2 -21437.743} C_VEL
LIN {X 0,Y 203.896,Z 668.02,A -85,B 0,C 180,E1 -21441.46,E2 -21441.46} C_VEL
LIN {X 0,Y 206.61,Z 658.357,A -85,B 0,C 180,E1 -21445.164,E2 -21445.164} C_VEL
LIN {X 0,Y 210.175,Z 646.326,A -85,B 0,C 180,E1 -21449.004,E2 -21449.004} C_VEL
LIN {X 0,Y 213.893,Z 634.018,A -85,B 0,C 180,E1 -21452.273,E2 -21452.273} C_VEL
LIN {X 0,Y 217.948,Z 620.798,A -85,B 0,C 180,E1 -21455.199,E2 -21455.199} C_VEL
LIN {X 0,Y 222.04,Z 606.432,A -85,B 0,C 180,E1 -21457.858,E2 -21457.858} C_VEL
LIN {X 0,Y 224.897,Z 595.699,A -85,B 0,C 180,E1 -21459.573,E2 -21459.573} C_VEL
LIN {X 0,Y 221.889,Z 586.073,A -85,B 0,C 180,E1 -21461.694,E2 -21461.694} C_VEL
LIN {X 0,Y 217.855,Z 574.778,A -85,B 0,C 180,E1 -21464.126,E2 -21464.126} C_VEL
LIN {X 0,Y 214.086,Z 565.197,A -85,B 0,C 180,E1 -21466.239,E2 -21466.239} C_VEL
LIN {X 0,Y 215.487,Z 565.529,A -85,B 0,C 180,E1 -21466.77,E2 -21466.77} C_VEL
LIN {X 0,Y 217.459,Z 564.612,A -85,B 0,C 180,E1 -21467.373,E2 -21467.373} C_VEL
LIN {X 0,Y 218.645,Z 564.986,A -85,B 0,C 180,E1 -21467.808,E2 -21467.808} C_VEL
LIN {X 0,Y 223.759,Z 574.084,A -85,B 0,C 180,E1 -21470.312,E2 -21470.312} C_VEL
LIN {X 0,Y 228.474,Z 583.768,A -85,B 0,C 180,E1 -21472.731,E2 -21472.731} C_VEL
LIN {X 0,Y 232.178,Z 593.302,A -85,B 0,C 180,E1 -21474.89,E2 -21474.89} C_VEL
LIN {X 0,Y 234.651,Z 602.435,A -85,B 0,C 180,E1 -21476.759,E2 -21476.759} C_VEL
LIN {X 0,Y 237.094,Z 615.96,A -85,B 0,C 180,E1 -21479.458,E2 -21479.458} C_VEL
LIN {X 0,Y 237.737,Z 620.761,A -85,B 0,C 180,E1 -21480.427,E2 -21480.427} C_VEL
LIN {X 0,Y 233.651,Z 634.438,A -85,B 0,C 180,E1 -21482.209,E2 -21482.209} C_VEL
LIN {X 0,Y 228.713,Z 648.78,A -85,B 0,C 180,E1 -21484.518,E2 -21484.518} C_VEL
LIN {X 0,Y 224.752,Z 658.985,A -85,B 0,C 180,E1 -21486.502,E2 -21486.502} C_VEL
LIN {X 0,Y 219.77,Z 671.335,A -85,B 0,C 180,E1 -21489.403,E2 -21489.403} C_VEL
LIN {X 0,Y 215.24,Z 681.878,A -85,B 0,C 180,E1 -21492.419,E2 -21492.419} C_VEL
LIN {X 0,Y 210.602,Z 692.041,A -85,B 0,C 180,E1 -21495.997,E2 -21495.997} C_VEL
LIN {X 0,Y 206.882,Z 700.431,A -85,B 0,C 180,E1 -21499.675,E2 -21499.675} C_VEL
LIN {X 0,Y 203.299,Z 708.453,A -85,B 0,C 180,E1 -21504.045,E2 -21504.045} C_VEL
LIN {X 0,Y 200.94,Z 714.195,A -85,B 0,C 180,E1 -21507.994,E2 -21507.994} C_VEL
LIN {X 0,Y 199.308,Z 718.77,A -85,B 0,C 180,E1 -21512.019,E2 -21512.019} C_VEL
LIN {X 0,Y 198.092,Z 722.637,A -85,B 0,C 180,E1 -21516.58,E2 -21516.58} C_VEL
LIN {X 0,Y 197.534,Z 724.867,A -85,B 0,C 180,E1 -21520.245,E2 -21520.245} C_VEL
LIN {X 0,Y 197.33,Z 726.388,A -85,B 0,C 180,E1 -21524.434,E2 -21524.434} C_VEL
LIN {X 0,Y 197.52,Z 727.017,A -85,B 0,C 180,E1 -21528.674,E2 -21528.674} C_VEL
LIN {X 0,Y 198.204,Z 726.561,A -85,B 0,C 180,E1 -21532.954,E2 -21532.954} C_VEL
LIN {X 0,Y 199.487,Z 725.134,A -85,B 0,C 180,E1 -21537.255,E2 -21537.255} C_VEL
LIN {X 0,Y 201.523,Z 722.619,A -85,B 0,C 180,E1 -21541.539,E2 -21541.539} C_VEL
LIN {X 0,Y 204.323,Z 718.936,A -85,B 0,C 180,E1 -21545.782,E2 -21545.782} C_VEL
LIN {X 0,Y 208.058,Z 714.072,A -85,B 0,C 180,E1 -21549.923,E2 -21549.923} C_VEL
LIN {X 0,Y 212.722,Z 707.872,A -85,B 0,C 180,E1 -21553.929,E2 -21553.929} C_VEL
LIN {X 0,Y 219.083,Z 699.11,A -85,B 0,C 180,E1 -21558.228,E2 -21558.228} C_VEL
LIN {X 0,Y 225.643,Z 689.481,A -85,B 0,C 180,E1 -21561.851,E2 -21561.851} C_VEL
LIN {X 0,Y 231.983,Z 679.353,A -85,B 0,C 180,E1 -21564.878,E2 -21564.878} C_VEL
LIN {X 0,Y 237.924,Z 669.194,A -85,B 0,C 180,E1 -21567.332,E2 -21567.332} C_VEL
LIN {X 0,Y 244.243,Z 657.356,A -85,B 0,C 180,E1 -21569.678,E2 -21569.678} C_VEL
LIN {X 0,Y 250.344,Z 644.537,A -85,B 0,C 180,E1 -21571.733,E2 -21571.733} C_VEL
LIN {X 0,Y 254.585,Z 634.513,A -85,B 0,C 180,E1 -21573.069,E2 -21573.069} C_VEL
LIN {X 0,Y 254.754,Z 633.381,A -85,B 0,C 180,E1 -21573.297,E2 -21573.297} C_VEL
LIN {X 0,Y 254.161,Z 625.373,A -85,B 0,C 180,E1 -21575.494,E2 -21575.494} C_VEL
LIN {X 0,Y 252.84,Z 618.954,A -85,B 0,C 180,E1 -21577.529,E2 -21577.529} C_VEL
LIN {X 0,Y 250.322,Z 610.629,A -85,B 0,C 180,E1 -21580.525,E2 -21580.525} C_VEL
LIN {X 0,Y 247.554,Z 603.527,A -85,B 0,C 180,E1 -21583.506,E2 -21583.506} C_VEL
LIN {X 0,Y 244.607,Z 597.005,A -85,B 0,C 180,E1 -21586.711,E2 -21586.711} C_VEL
LIN {X 0,Y 242.531,Z 592.619,A -85,B 0,C 180,E1 -21589.142,E2 -21589.142} C_VEL
LIN {X 0,Y 240.307,Z 588.632,A -85,B 0,C 180,E1 -21591.908,E2 -21591.908} C_VEL
LIN {X 0,Y 237.411,Z 583.604,A -85,B 0,C 180,E1 -21596.4,E2 -21596.4} C_VEL
LIN {X 0,Y 234.92,Z 579.491,A -85,B 0,C 180,E1 -21602.571,E2 -21602.571} C_VEL
LIN {X 0,Y 234.259,Z 579.587,A -85,B 0,C 180,E1 -21608.626,E2 -21608.626} C_VEL
LIN {X 0,Y 235.559,Z 581.397,A -85,B 0,C 180,E1 -21614.028,E2 -21614.028} C_VEL
LIN {X 0,Y 237.224,Z 584.568,A -85,B 0,C 180,E1 -21617.677,E2 -21617.677} C_VEL
LIN {X 0,Y 240.665,Z 589.452,A -85,B 0,C 180,E1 -21622.31,E2 -21622.31} C_VEL
LIN {X 0,Y 242.773,Z 593.691,A -85,B 0,C 180,E1 -21624.819,E2 -21624.819} C_VEL
LIN {X 0,Y 245.265,Z 600.544,A -85,B 0,C 180,E1 -21627.751,E2 -21627.751} C_VEL
LIN {X 0,Y 247.099,Z 606.148,A -85,B 0,C 180,E1 -21629.849,E2 -21629.849} C_VEL
LIN {X 0,Y 250.161,Z 616.238,A -85,B 0,C 180,E1 -21633.218,E2 -21633.218} C_VEL
LIN {X 0,Y 251.537,Z 622.294,A -85,B 0,C 180,E1 -21634.943,E2 -21634.943} C_VEL
LIN {X 0,Y 251.837,Z 626.377,A -85,B 0,C 180,E1 -21635.876,E2 -21635.876} C_VEL
LIN {X 0,Y 250.933,Z 639.809,A -85,B 0,C 180,E1 -21638.356,E2 -21638.356} C_VEL
LIN {X 0,Y 249.392,Z 650.1,A -85,B 0,C 180,E1 -21640.22,E2 -21640.22} C_VEL
LIN {X 0,Y 247.129,Z 661.287,A -85,B 0,C 180,E1 -21642.314,E2 -21642.314} C_VEL
LIN {X 0,Y 246.071,Z 664.349,A -85,B 0,C 180,E1 -21642.806,E2 -21642.806} C_VEL
LIN {X 0,Y 244.359,Z 667.48,A -85,B 0,C 180,E1 -21643.17,E2 -21643.17} C_VEL
LIN {X 0,Y 239.807,Z 673.638,A -85,B 0,C 180,E1 -21643.671,E2 -21643.671} C_VEL
LIN {X 0,Y 233.521,Z 681.164,A -85,B 0,C 180,E1 -21644.322,E2 -21644.322} C_VEL
LIN {X 0,Y 230.479,Z 685.529,A -85,B 0,C 180,E1 -21645.016,E2 -21645.016} C_VEL
LIN {X 0,Y 223.868,Z 696.873,A -85,B 0,C 180,E1 -21647.552,E2 -21647.552} C_VEL
LIN {X 0,Y 216.712,Z 708.301,A -85,B 0,C 180,E1 -21650.777,E2 -21650.777} C_VEL
LIN {X 0,Y 210.414,Z 717.946,A -85,B 0,C 180,E1 -21654.234,E2 -21654.234} C_VEL
LIN {X 0,Y 204.791,Z 726.113,A -85,B 0,C 180,E1 -21657.867,E2 -21657.867} C_VEL
LIN {X 0,Y 200.043,Z 733.172,A -85,B 0,C 180,E1 -21661.822,E2 -21661.822} C_VEL
LIN {X 0,Y 195.691,Z 739.873,A -85,B 0,C 180,E1 -21666.734,E2 -21666.734} C_VEL
LIN {X 0,Y 192.957,Z 744.466,A -85,B 0,C 180,E1 -21671.258,E2 -21671.258} C_VEL
LIN {X 0,Y 191.459,Z 747.452,A -85,B 0,C 180,E1 -21675.113,E2 -21675.113} C_VEL
LIN {X 0,Y 190.557,Z 749.7,A -85,B 0,C 180,E1 -21679.376,E2 -21679.376} C_VEL
LIN {X 0,Y 190.497,Z 751.073,A -85,B 0,C 180,E1 -21683.648,E2 -21683.648} C_VEL
LIN {X 0,Y 190.659,Z 751.375,A -85,B 0,C 180,E1 -21687.89,E2 -21687.89} C_VEL
LIN {X 0,Y 190.75,Z 751.186,A -85,B 0,C 180,E1 -21690.002,E2 -21690.002} C_VEL
LIN {X 0,Y 190.701,Z 750.73,A -85,B 0,C 180,E1 -21692.114,E2 -21692.114} C_VEL
LIN {X 0,Y 190.603,Z 748.943,A -85,B 0,C 180,E1 -21696.353,E2 -21696.353} C_VEL
LIN {X 0,Y 190.677,Z 746.161,A -85,B 0,C 180,E1 -21700.622,E2 -21700.622} C_VEL
LIN {X 0,Y 191.83,Z 741.083,A -85,B 0,C 180,E1 -21705.951,E2 -21705.951} C_VEL
LIN {X 0,Y 193.561,Z 735.653,A -85,B 0,C 180,E1 -21710.18,E2 -21710.18} C_VEL
LIN {X 0,Y 194.432,Z 733.433,A -85,B 0,C 180,E1 -21711.748,E2 -21711.748} C_VEL
LIN {X 0,Y 198.874,Z 728.074,A -85,B 0,C 180,E1 -21717.351,E2 -21717.351} C_VEL
LIN {X 0,Y 205.983,Z 720.868,A -85,B 0,C 180,E1 -21723.089,E2 -21723.089} C_VEL
LIN {X 0,Y 216.778,Z 711.175,A -85,B 0,C 180,E1 -21728.915,E2 -21728.915} C_VEL
LIN {X 0,Y 229.117,Z 700.907,A -85,B 0,C 180,E1 -21733.646,E2 -21733.646} C_VEL
LIN {X 0,Y 243.066,Z 689.992,A -85,B 0,C 180,E1 -21737.504,E2 -21737.504} C_VEL
LIN {X 0,Y 245.564,Z 688.069,A -85,B 0,C 180,E1 -21738.085,E2 -21738.085} C_VEL
LIN {X 0,Y 245.994,Z 687.547,A -85,B 0,C 180,E1 -21738.549,E2 -21738.549} C_VEL
LIN {X 0,Y 234.118,Z 693.567,A -85,B 0,C 180,E1 -21742.021,E2 -21742.021} C_VEL
LIN {X 0,Y 224.195,Z 698.216,A -85,B 0,C 180,E1 -21745.65,E2 -21745.65} C_VEL
LIN {X 0,Y 214.067,Z 702.603,A -85,B 0,C 180,E1 -21750.498,E2 -21750.498} C_VEL
LIN {X 0,Y 205.876,Z 705.515,A -85,B 0,C 180,E1 -21755.818,E2 -21755.818} C_VEL
LIN {X 0,Y 199.631,Z 706.878,A -85,B 0,C 180,E1 -21761.529,E2 -21761.529} C_VEL
LIN {X 0,Y 195.434,Z 706.56,A -85,B 0,C 180,E1 -21767.54,E2 -21767.54} C_VEL
LIN {X 0,Y 193.588,Z 705.373,A -85,B 0,C 180,E1 -21771.651,E2 -21771.651} C_VEL
LIN {X 0,Y 192.225,Z 703.397,A -85,B 0,C 180,E1 -21775.808,E2 -21775.808} C_VEL
LIN {X 0,Y 191.682,Z 700.501,A -85,B 0,C 180,E1 -21780.001,E2 -21780.001} C_VEL
LIN {X 0,Y 191.74,Z 696.69,A -85,B 0,C 180,E1 -21784.205,E2 -21784.205} C_VEL
LIN {X 0,Y 192.182,Z 691.01,A -85,B 0,C 180,E1 -21789.104,E2 -21789.104} C_VEL
LIN {X 0,Y 193.127,Z 684.295,A -85,B 0,C 180,E1 -21793.683,E2 -21793.683} C_VEL
LIN {X 0,Y 194.963,Z 675.78,A -85,B 0,C 180,E1 -21798.387,E2 -21798.387} C_VEL
LIN {X 0,Y 197.369,Z 666.759,A -85,B 0,C 180,E1 -21802.488,E2 -21802.488} C_VEL
LIN {X 0,Y 200.493,Z 656.035,A -85,B 0,C 180,E1 -21806.548,E2 -21806.548} C_VEL
LIN {X 0,Y 203.848,Z 645.17,A -85,B 0,C 180,E1 -21809.984,E2 -21809.984} C_VEL
LIN {X 0,Y 207.763,Z 632.529,A -85,B 0,C 180,E1 -21813.347,E2 -21813.347} C_VEL
LIN {X 0,Y 212.029,Z 619.019,A -85,B 0,C 180,E1 -21816.335,E2 -21816.335} C_VEL
LIN {X 0,Y 216.515,Z 603.712,A -85,B 0,C 180,E1 -21819.15,E2 -21819.15} C_VEL
LIN {X 0,Y 218.104,Z 597.686,A -85,B 0,C 180,E1 -21820.127,E2 -21820.127} C_VEL
LIN {X 0,Y 217.422,Z 594.512,A -85,B 0,C 180,E1 -21820.818,E2 -21820.818} C_VEL
LIN {X 0,Y 212.956,Z 581.128,A -85,B 0,C 180,E1 -21823.873,E2 -21823.873} C_VEL
LIN {X 0,Y 210.105,Z 573.51,A -85,B 0,C 180,E1 -21825.623,E2 -21825.623} C_VEL
LIN {X 0,Y 211.24,Z 573.927,A -85,B 0,C 180,E1 -21826.098,E2 -21826.098} C_VEL
LIN {X 0,Y 213.174,Z 573.267,A -85,B 0,C 180,E1 -21826.729,E2 -21826.729} C_VEL
LIN {X 0,Y 214.411,Z 572.432,A -85,B 0,C 180,E1 -21827.076,E2 -21827.076} C_VEL
LIN {X 0,Y 215.971,Z 572.204,A -85,B 0,C 180,E1 -21827.595,E2 -21827.595} C_VEL
LIN {X 0,Y 220.389,Z 580.705,A -85,B 0,C 180,E1 -21830.002,E2 -21830.002} C_VEL
LIN {X 0,Y 223.56,Z 587.618,A -85,B 0,C 180,E1 -21831.807,E2 -21831.807} C_VEL
LIN {X 0,Y 227.239,Z 597.582,A -85,B 0,C 180,E1 -21834.202,E2 -21834.202} C_VEL
LIN {X 0,Y 229.195,Z 605.403,A -85,B 0,C 180,E1 -21835.887,E2 -21835.887} C_VEL
LIN {X 0,Y 231.185,Z 617.243,A -85,B 0,C 180,E1 -21838.344,E2 -21838.344} C_VEL
LIN {X 0,Y 231.751,Z 623.25,A -85,B 0,C 180,E1 -21839.584,E2 -21839.584} C_VEL
LIN {X 0,Y 227.045,Z 637.838,A -85,B 0,C 180,E1 -21841.579,E2 -21841.579} C_VEL
LIN {X 0,Y 222.371,Z 650.685,A -85,B 0,C 180,E1 -21843.737,E2 -21843.737} C_VEL
LIN {X 0,Y 217.602,Z 662.611,A -85,B 0,C 180,E1 -21846.187,E2 -21846.187} C_VEL
LIN {X 0,Y 212.521,Z 674.445,A -85,B 0,C 180,E1 -21849.174,E2 -21849.174} C_VEL
LIN {X 0,Y 207.941,Z 684.55,A -85,B 0,C 180,E1 -21852.289,E2 -21852.289} C_VEL
LIN {X 0,Y 203.764,Z 693.296,A -85,B 0,C 180,E1 -21855.517,E2 -21855.517} C_VEL
LIN {X 0,Y 199.431,Z 702.641,A -85,B 0,C 180,E1 -21859.849,E2 -21859.849} C_VEL
LIN {X 0,Y 196.252,Z 709.448,A -85,B 0,C 180,E1 -21863.831,E2 -21863.831} C_VEL
LIN {X 0,Y 193.842,Z 715.068,A -85,B 0,C 180,E1 -21867.92,E2 -21867.92} C_VEL
LIN {X 0,Y 192.159,Z 719.59,A -85,B 0,C 180,E1 -21872.094,E2 -21872.094} C_VEL
LIN {X 0,Y 191.015,Z 723.168,A -85,B 0,C 180,E1 -21876.573,E2 -21876.573} C_VEL
LIN {X 0,Y 190.407,Z 725.501,A -85,B 0,C 180,E1 -21880.633,E2 -21880.633} C_VEL
LIN {X 0,Y 190.295,Z 727.213,A -85,B 0,C 180,E1 -21886.209,E2 -21886.209} C_VEL
LIN {X 0,Y 190.835,Z 727.355,A -85,B 0,C 180,E1 -21891.607,E2 -21891.607} C_VEL
LIN {X 0,Y 191.953,Z 726.301,A -85,B 0,C 180,E1 -21896.06,E2 -21896.06} C_VEL
LIN {X 0,Y 193.83,Z 724.259,A -85,B 0,C 180,E1 -21900.502,E2 -21900.502} C_VEL
LIN {X 0,Y 196.487,Z 721.074,A -85,B 0,C 180,E1 -21904.907,E2 -21904.907} C_VEL
LIN {X 0,Y 200.343,Z 716.363,A -85,B 0,C 180,E1 -21909.487,E2 -21909.487} C_VEL
LIN {X 0,Y 205.525,Z 709.899,A -85,B 0,C 180,E1 -21914.101,E2 -21914.101} C_VEL
LIN {X 0,Y 210.965,Z 702.915,A -85,B 0,C 180,E1 -21917.897,E2 -21917.897} C_VEL
LIN {X 0,Y 216.536,Z 695.354,A -85,B 0,C 180,E1 -21921.161,E2 -21921.161} C_VEL
LIN {X 0,Y 222.797,Z 686.232,A -85,B 0,C 180,E1 -21924.314,E2 -21924.314} C_VEL
LIN {X 0,Y 229.692,Z 675.456,A -85,B 0,C 180,E1 -21927.287,E2 -21927.287} C_VEL
LIN {X 0,Y 236.578,Z 663.621,A -85,B 0,C 180,E1 -21929.902,E2 -21929.902} C_VEL
LIN {X 0,Y 242.62,Z 652.13,A -85,B 0,C 180,E1 -21931.963,E2 -21931.963} C_VEL
LIN {X 0,Y 248.61,Z 639.242,A -85,B 0,C 180,E1 -21933.832,E2 -21933.832} C_VEL
LIN {X 0,Y 249.726,Z 636.495,A -85,B 0,C 180,E1 -21934.228,E2 -21934.228} C_VEL
LIN {X 0,Y 249.328,Z 629.03,A -85,B 0,C 180,E1 -21936.394,E2 -21936.394} C_VEL
LIN {X 0,Y 248.207,Z 623.081,A -85,B 0,C 180,E1 -21938.401,E2 -21938.401} C_VEL
LIN {X 0,Y 245.869,Z 614.55,A -85,B 0,C 180,E1 -21941.673,E2 -21941.673} C_VEL
LIN {X 0,Y 243.233,Z 607.349,A -85,B 0,C 180,E1 -21944.926,E2 -21944.926} C_VEL
LIN {X 0,Y 240.019,Z 599.844,A -85,B 0,C 180,E1 -21949.027,E2 -21949.027} C_VEL
LIN {X 0,Y 237.666,Z 594.944,A -85,B 0,C 180,E1 -21952.352,E2 -21952.352} C_VEL
LIN {X 0,Y 235.122,Z 590.192,A -85,B 0,C 180,E1 -21956.786,E2 -21956.786} C_VEL
LIN {X 0,Y 233.148,Z 586.368,A -85,B 0,C 180,E1 -21962.591,E2 -21962.591} C_VEL
LIN {X 0,Y 232.555,Z 586.478,A -85,B 0,C 180,E1 -21968.69,E2 -21968.69} C_VEL
LIN {X 0,Y 233.863,Z 588.385,A -85,B 0,C 180,E1 -21974.132,E2 -21974.132} C_VEL
LIN {X 0,Y 237.821,Z 595.206,A -85,B 0,C 180,E1 -21981.336,E2 -21981.336} C_VEL
LIN {X 0,Y 240.021,Z 599.697,A -85,B 0,C 180,E1 -21984.2,E2 -21984.2} C_VEL
LIN {X 0,Y 242.847,Z 608.558,A -85,B 0,C 180,E1 -21988.051,E2 -21988.051} C_VEL
LIN {X 0,Y 245.989,Z 620.174,A -85,B 0,C 180,E1 -21992.163,E2 -21992.163} C_VEL
LIN {X 0,Y 247.273,Z 626.95,A -85,B 0,C 180,E1 -21994.197,E2 -21994.197} C_VEL
LIN {X 0,Y 247.401,Z 630.098,A -85,B 0,C 180,E1 -21994.929,E2 -21994.929} C_VEL
LIN {X 0,Y 245.948,Z 644.003,A -85,B 0,C 180,E1 -21997.616,E2 -21997.616} C_VEL
LIN {X 0,Y 243.68,Z 655.641,A -85,B 0,C 180,E1 -21999.784,E2 -21999.784} C_VEL
LIN {X 0,Y 241.923,Z 663.15,A -85,B 0,C 180,E1 -22001.267,E2 -22001.267} C_VEL
LIN {X 0,Y 235.724,Z 675.746,A -85,B 0,C 180,E1 -22003.204,E2 -22003.204} C_VEL
LIN {X 0,Y 230.479,Z 685.529,A -85,B 0,C 180,E1 -22005.016,E2 -22005.016} C_VEL
LIN {X 0,Y 227.612,Z 689.787,A -85,B 0,C 180,E1 -22005.785,E2 -22005.785} C_VEL
LIN {X 0,Y 221.57,Z 696.518,A -85,B 0,C 180,E1 -22006.83,E2 -22006.83} C_VEL
LIN {X 0,Y 215.457,Z 702.868,A -85,B 0,C 180,E1 -22007.993,E2 -22007.993} C_VEL
LIN {X 0,Y 212.522,Z 706.447,A -85,B 0,C 180,E1 -22008.945,E2 -22008.945} C_VEL
LIN {X 0,Y 206.192,Z 715.71,A -85,B 0,C 180,E1 -22012.158,E2 -22012.158} C_VEL
LIN {X 0,Y 200.093,Z 724.178,A -85,B 0,C 180,E1 -22015.81,E2 -22015.81} C_VEL
LIN {X 0,Y 194.419,Z 731.999,A -85,B 0,C 180,E1 -22020.175,E2 -22020.175} C_VEL
LIN {X 0,Y 189.918,Z 738.382,A -85,B 0,C 180,E1 -22024.817,E2 -22024.817} C_VEL
LIN {X 0,Y 186.342,Z 743.851,A -85,B 0,C 180,E1 -22030.16,E2 -22030.16} C_VEL
LIN {X 0,Y 184.531,Z 747.123,A -85,B 0,C 180,E1 -22034.541,E2 -22034.541} C_VEL
LIN {X 0,Y 183.497,Z 749.318,A -85,B 0,C 180,E1 -22038.962,E2 -22038.962} C_VEL
LIN {X 0,Y 183.391,Z 750.652,A -85,B 0,C 180,E1 -22043.401,E2 -22043.401} C_VEL
LIN {X 0,Y 183.589,Z 750.909,A -85,B 0,C 180,E1 -22047.808,E2 -22047.808} C_VEL
LIN {X 0,Y 183.679,Z 750.691,A -85,B 0,C 180,E1 -22050.002,E2 -22050.002} C_VEL
LIN {X 0,Y 183.632,Z 750.226,A -85,B 0,C 180,E1 -22052.196,E2 -22052.196} C_VEL
LIN {X 0,Y 183.513,Z 748.386,A -85,B 0,C 180,E1 -22056.6,E2 -22056.6} C_VEL
LIN {X 0,Y 183.651,Z 745.541,A -85,B 0,C 180,E1 -22061.033,E2 -22061.033} C_VEL
LIN {X 0,Y 184.579,Z 741.54,A -85,B 0,C 180,E1 -22065.46,E2 -22065.46} C_VEL
LIN {X 0,Y 186.231,Z 736.394,A -85,B 0,C 180,E1 -22069.857,E2 -22069.857} C_VEL
LIN {X 0,Y 187.402,Z 733.427,A -85,B 0,C 180,E1 -22072.028,E2 -22072.028} C_VEL
LIN {X 0,Y 192.499,Z 727.981,A -85,B 0,C 180,E1 -22078.337,E2 -22078.337} C_VEL
LIN {X 0,Y 200.028,Z 721.128,A -85,B 0,C 180,E1 -22084.207,E2 -22084.207} C_VEL
LIN {X 0,Y 211.213,Z 712.075,A -85,B 0,C 180,E1 -22090.066,E2 -22090.066} C_VEL
LIN {X 0,Y 224.147,Z 702.347,A -85,B 0,C 180,E1 -22094.87,E2 -22094.87} C_VEL
LIN {X 0,Y 236,Z 693.857,A -85,B 0,C 180,E1 -22098.117,E2 -22098.117} C_VEL
LIN {X 0,Y 236.731,Z 693.11,A -85,B 0,C 180,E1 -22098.751,E2 -22098.751} C_VEL
LIN {X 0,Y 222.671,Z 699.173,A -85,B 0,C 180,E1 -22103.154,E2 -22103.154} C_VEL
LIN {X 0,Y 211.514,Z 703.503,A -85,B 0,C 180,E1 -22107.885,E2 -22107.885} C_VEL
LIN {X 0,Y 202.208,Z 706.475,A -85,B 0,C 180,E1 -22113.14,E2 -22113.14} C_VEL
LIN {X 0,Y 197.218,Z 707.679,A -85,B 0,C 180,E1 -22116.922,E2 -22116.922} C_VEL
LIN {X 0,Y 191.29,Z 708.145,A -85,B 0,C 180,E1 -22122.908,E2 -22122.908} C_VEL
LIN {X 0,Y 187.542,Z 706.918,A -85,B 0,C 180,E1 -22129.202,E2 -22129.202} C_VEL
LIN {X 0,Y 185.828,Z 705.142,A -85,B 0,C 180,E1 -22133.486,E2 -22133.486} C_VEL
LIN {X 0,Y 184.807,Z 702.529,A -85,B 0,C 180,E1 -22137.822,E2 -22137.822} C_VEL
LIN {X 0,Y 184.558,Z 698.993,A -85,B 0,C 180,E1 -22142.183,E2 -22142.183} C_VEL
LIN {X 0,Y 184.759,Z 694.501,A -85,B 0,C 180,E1 -22146.554,E2 -22146.554} C_VEL
LIN {X 0,Y 185.343,Z 688.964,A -85,B 0,C 180,E1 -22150.93,E2 -22150.93} C_VEL
LIN {X 0,Y 186.494,Z 682.222,A -85,B 0,C 180,E1 -22155.296,E2 -22155.296} C_VEL
LIN {X 0,Y 188.406,Z 674.186,A -85,B 0,C 180,E1 -22159.617,E2 -22159.617} C_VEL
LIN {X 0,Y 190.771,Z 665.826,A -85,B 0,C 180,E1 -22163.413,E2 -22163.413} C_VEL
LIN {X 0,Y 194.033,Z 655.044,A -85,B 0,C 180,E1 -22167.505,E2 -22167.505} C_VEL
LIN {X 0,Y 197.936,Z 642.666,A -85,B 0,C 180,E1 -22171.419,E2 -22171.419} C_VEL
LIN {X 0,Y 201.715,Z 630.969,A -85,B 0,C 180,E1 -22174.485,E2 -22174.485} C_VEL
LIN {X 0,Y 206.155,Z 617.046,A -85,B 0,C 180,E1 -22177.545,E2 -22177.545} C_VEL
LIN {X 0,Y 210.63,Z 602.083,A -85,B 0,C 180,E1 -22180.278,E2 -22180.278} C_VEL
LIN {X 0,Y 211.475,Z 598.897,A -85,B 0,C 180,E1 -22180.81,E2 -22180.81} C_VEL
LIN {X 0,Y 207.013,Z 584.881,A -85,B 0,C 180,E1 -22184.16,E2 -22184.16} C_VEL
LIN {X 0,Y 205.839,Z 581.594,A -85,B 0,C 180,E1 -22184.989,E2 -22184.989} C_VEL
LIN {X 0,Y 206.954,Z 582.035,A -85,B 0,C 180,E1 -22185.493,E2 -22185.493} C_VEL
LIN {X 0,Y 208.961,Z 581.401,A -85,B 0,C 180,E1 -22186.172,E2 -22186.172} C_VEL
LIN {X 0,Y 209.988,Z 580.76,A -85,B 0,C 180,E1 -22186.468,E2 -22186.468} C_VEL
LIN {X 0,Y 213.775,Z 580.53,A -85,B 0,C 180,E1 -22187.795,E2 -22187.795} C_VEL
LIN {X 0,Y 218.806,Z 591.737,A -85,B 0,C 180,E1 -22190.951,E2 -22190.951} C_VEL
LIN {X 0,Y 222.517,Z 602.519,A -85,B 0,C 180,E1 -22193.648,E2 -22193.648} C_VEL
LIN {X 0,Y 224.621,Z 613.241,A -85,B 0,C 180,E1 -22196.034,E2 -22196.034} C_VEL
LIN {X 0,Y 225.939,Z 623.701,A -85,B 0,C 180,E1 -22198.33,E2 -22198.33} C_VEL
LIN {X 0,Y 225.946,Z 625,A -85,B 0,C 180,E1 -22198.586,E2 -22198.586} C_VEL
LIN {X 0,Y 221.351,Z 638.721,A -85,B 0,C 180,E1 -22200.517,E2 -22200.517} C_VEL
LIN {X 0,Y 216.079,Z 652.546,A -85,B 0,C 180,E1 -22202.911,E2 -22202.911} C_VEL
LIN {X 0,Y 211.2,Z 664.321,A -85,B 0,C 180,E1 -22205.419,E2 -22205.419} C_VEL
LIN {X 0,Y 205.968,Z 675.971,A -85,B 0,C 180,E1 -22208.479,E2 -22208.479} C_VEL
LIN {X 0,Y 201.25,Z 685.896,A -85,B 0,C 180,E1 -22211.68,E2 -22211.68} C_VEL
LIN {X 0,Y 196.94,Z 694.491,A -85,B 0,C 180,E1 -22215.004,E2 -22215.004} C_VEL
LIN {X 0,Y 193.398,Z 701.791,A -85,B 0,C 180,E1 -22218.469,E2 -22218.469} C_VEL
LIN {X 0,Y 189.929,Z 708.853,A -85,B 0,C 180,E1 -22222.556,E2 -22222.556} C_VEL
LIN {X 0,Y 187.29,Z 714.708,A -85,B 0,C 180,E1 -22226.771,E2 -22226.771} C_VEL
LIN {X 0,Y 185.015,Z 720.384,A -85,B 0,C 180,E1 -22232.175,E2 -22232.175} C_VEL
LIN {X 0,Y 183.909,Z 723.706,A -85,B 0,C 180,E1 -22236.581,E2 -22236.581} C_VEL
LIN {X 0,Y 183.273,Z 726.097,A -85,B 0,C 180,E1 -22241.052,E2 -22241.052} C_VEL
LIN {X 0,Y 183.192,Z 727.479,A -85,B 0,C 180,E1 -22245.575,E2 -22245.575} C_VEL
LIN {X 0,Y 183.497,Z 727.897,A -85,B 0,C 180,E1 -22250.161,E2 -22250.161} C_VEL
LIN {X 0,Y 184.447,Z 727.337,A -85,B 0,C 180,E1 -22254.777,E2 -22254.777} C_VEL
LIN {X 0,Y 186.367,Z 725.466,A -85,B 0,C 180,E1 -22259.847,E2 -22259.847} C_VEL
LIN {X 0,Y 189.625,Z 721.904,A -85,B 0,C 180,E1 -22265.373,E2 -22265.373} C_VEL
LIN {X 0,Y 193.025,Z 718.08,A -85,B 0,C 180,E1 -22269.463,E2 -22269.463} C_VEL
LIN {X 0,Y 197.789,Z 712.563,A -85,B 0,C 180,E1 -22273.856,E2 -22273.856} C_VEL
LIN {X 0,Y 203.448,Z 705.717,A -85,B 0,C 180,E1 -22277.959,E2 -22277.959} C_VEL
LIN {X 0,Y 210.02,Z 697.331,A -85,B 0,C 180,E1 -22281.845,E2 -22281.845} C_VEL
LIN {X 0,Y 216.469,Z 688.55,A -85,B 0,C 180,E1 -22285.058,E2 -22285.058} C_VEL
LIN {X 0,Y 223.548,Z 678.169,A -85,B 0,C 180,E1 -22288.081,E2 -22288.081} C_VEL
LIN {X 0,Y 231.264,Z 665.573,A -85,B 0,C 180,E1 -22290.975,E2 -22290.975} C_VEL
LIN {X 0,Y 237.812,Z 653.581,A -85,B 0,C 180,E1 -22293.161,E2 -22293.161} C_VEL
LIN {X 0,Y 244.318,Z 640.16,A -85,B 0,C 180,E1 -22295.129,E2 -22295.129} C_VEL
LIN {X 0,Y 244.687,Z 638.526,A -85,B 0,C 180,E1 -22295.491,E2 -22295.491} C_VEL
LIN {X 0,Y 244.421,Z 632.265,A -85,B 0,C 180,E1 -22297.44,E2 -22297.44} C_VEL
LIN {X 0,Y 243.076,Z 624.943,A -85,B 0,C 180,E1 -22300.139,E2 -22300.139} C_VEL
LIN {X 0,Y 241.23,Z 617.987,A -85,B 0,C 180,E1 -22303.061,E2 -22303.061} C_VEL
LIN {X 0,Y 238.924,Z 611.234,A -85,B 0,C 180,E1 -22306.389,E2 -22306.389} C_VEL
LIN {X 0,Y 236.705,Z 605.497,A -85,B 0,C 180,E1 -22309.737,E2 -22309.737} C_VEL
LIN {X 0,Y 234.687,Z 600.891,A -85,B 0,C 180,E1 -22313.12,E2 -22313.12} C_VEL
LIN {X 0,Y 232.954,Z 597.224,A -85,B 0,C 180,E1 -22316.54,E2 -22316.54} C_VEL
LIN {X 0,Y 231.098,Z 593.23,A -85,B 0,C 180,E1 -22322.614,E2 -22322.614} C_VEL
LIN {X 0,Y 230.505,Z 593.179,A -85,B 0,C 180,E1 -22327.885,E2 -22327.885} C_VEL
LIN {X 0,Y 231.409,Z 594.648,A -85,B 0,C 180,E1 -22332.943,E2 -22332.943} C_VEL
LIN {X 0,Y 232.072,Z 595.907,A -85,B 0,C 180,E1 -22334.916,E2 -22334.916} C_VEL
LIN {X 0,Y 235.336,Z 601.694,A -85,B 0,C 180,E1 -22340.999,E2 -22340.999} C_VEL
LIN {X 0,Y 237.065,Z 605.633,A -85,B 0,C 180,E1 -22343.59,E2 -22343.59} C_VEL
LIN {X 0,Y 239.504,Z 614.451,A -85,B 0,C 180,E1 -22347.526,E2 -22347.526} C_VEL
LIN {X 0,Y 242.002,Z 625.339,A -85,B 0,C 180,E1 -22351.515,E2 -22351.515} C_VEL
LIN {X 0,Y 242.973,Z 632.206,A -85,B 0,C 180,E1 -22353.616,E2 -22353.616} C_VEL
LIN {X 0,Y 241.922,Z 641.767,A -85,B 0,C 180,E1 -22355.573,E2 -22355.573} C_VEL
LIN {X 0,Y 240.322,Z 650.951,A -85,B 0,C 180,E1 -22357.399,E2 -22357.399} C_VEL
LIN {X 0,Y 236.786,Z 664.846,A -85,B 0,C 180,E1 -22360.161,E2 -22360.161} C_VEL
LIN {X 0,Y 229.739,Z 678.345,A -85,B 0,C 180,E1 -22362.299,E2 -22362.299} C_VEL
LIN {X 0,Y 222.659,Z 690.637,A -85,B 0,C 180,E1 -22364.753,E2 -22364.753} C_VEL
LIN {X 0,Y 215.758,Z 701.514,A -85,B 0,C 180,E1 -22367.479,E2 -22367.479} C_VEL
LIN {X 0,Y 212.522,Z 706.447,A -85,B 0,C 180,E1 -22368.945,E2 -22368.945} C_VEL
LIN {X 0,Y 209.575,Z 710.016,A -85,B 0,C 180,E1 -22369.959,E2 -22369.959} C_VEL
LIN {X 0,Y 198.388,Z 719.76,A -85,B 0,C 180,E1 -22372.765,E2 -22372.765} C_VEL
LIN {X 0,Y 195.315,Z 722.699,A -85,B 0,C 180,E1 -22373.948,E2 -22373.948} C_VEL
LIN {X 0,Y 194.528,Z 723.654,A -85,B 0,C 180,E1 -22374.396,E2 -22374.396} C_VEL
LIN {X 0,Y 188.781,Z 731.085,A -85,B 0,C 180,E1 -22378.591,E2 -22378.591} C_VEL
LIN {X 0,Y 184.353,Z 736.903,A -85,B 0,C 180,E1 -22382.779,E2 -22382.779} C_VEL
LIN {X 0,Y 180.909,Z 741.625,A -85,B 0,C 180,E1 -22387.143,E2 -22387.143} C_VEL
LIN {X 0,Y 178.479,Z 745.282,A -85,B 0,C 180,E1 -22391.641,E2 -22391.641} C_VEL
LIN {X 0,Y 176.883,Z 747.983,A -85,B 0,C 180,E1 -22396.211,E2 -22396.211} C_VEL
LIN {X 0,Y 176.275,Z 749.682,A -85,B 0,C 180,E1 -22400.826,E2 -22400.826} C_VEL
LIN {X 0,Y 176.39,Z 750.459,A -85,B 0,C 180,E1 -22405.432,E2 -22405.432} C_VEL
LIN {X 0,Y 176.609,Z 750.194,A -85,B 0,C 180,E1 -22410.002,E2 -22410.002} C_VEL
LIN {X 0,Y 176.564,Z 749.702,A -85,B 0,C 180,E1 -22412.284,E2 -22412.284} C_VEL
LIN {X 0,Y 176.497,Z 748.529,A -85,B 0,C 180,E1 -22415.457,E2 -22415.457} C_VEL
LIN {X 0,Y 176.412,Z 746.489,A -85,B 0,C 180,E1 -22419.172,E2 -22419.172} C_VEL
LIN {X 0,Y 177.007,Z 743.058,A -85,B 0,C 180,E1 -22423.784,E2 -22423.784} C_VEL
LIN {X 0,Y 178.448,Z 738.407,A -85,B 0,C 180,E1 -22428.367,E2 -22428.367} C_VEL
LIN {X 0,Y 180.704,Z 732.915,A -85,B 0,C 180,E1 -22432.89,E2 -22432.89} C_VEL
LIN {X 0,Y 186.168,Z 727.813,A -85,B 0,C 180,E1 -22439.393,E2 -22439.393} C_VEL
LIN {X 0,Y 194.144,Z 721.417,A -85,B 0,C 180,E1 -22445.396,E2 -22445.396} C_VEL
LIN {X 0,Y 205.799,Z 712.976,A -85,B 0,C 180,E1 -22451.298,E2 -22451.298} C_VEL
LIN {X 0,Y 216.999,Z 705.252,A -85,B 0,C 180,E1 -22455.442,E2 -22455.442} C_VEL
LIN {X 0,Y 226.471,Z 699.034,A -85,B 0,C 180,E1 -22458.142,E2 -22458.142} C_VEL
LIN {X 0,Y 227.454,Z 698.116,A -85,B 0,C 180,E1 -22458.957,E2 -22458.957} C_VEL
LIN {X 0,Y 217.461,Z 701.891,A -85,B 0,C 180,E1 -22462.118,E2 -22462.118} C_VEL
LIN {X 0,Y 205.835,Z 705.71,A -85,B 0,C 180,E1 -22466.887,E2 -22466.887} C_VEL
LIN {X 0,Y 196.115,Z 708.278,A -85,B 0,C 180,E1 -22472.234,E2 -22472.234} C_VEL
LIN {X 0,Y 188.519,Z 709.389,A -85,B 0,C 180,E1 -22478.113,E2 -22478.113} C_VEL
LIN {X 0,Y 183.048,Z 708.953,A -85,B 0,C 180,E1 -22484.411,E2 -22484.411} C_VEL
LIN {X 0,Y 180.625,Z 707.719,A -85,B 0,C 180,E1 -22488.783,E2 -22488.783} C_VEL
LIN {X 0,Y 178.819,Z 705.774,A -85,B 0,C 180,E1 -22493.23,E2 -22493.23} C_VEL
LIN {X 0,Y 177.736,Z 702.913,A -85,B 0,C 180,E1 -22497.735,E2 -22497.735} C_VEL
LIN {X 0,Y 177.465,Z 699.235,A -85,B 0,C 180,E1 -22502.271,E2 -22502.271} C_VEL
LIN {X 0,Y 177.692,Z 694.51,A -85,B 0,C 180,E1 -22506.815,E2 -22506.815} C_VEL
LIN {X 0,Y 178.332,Z 688.782,A -85,B 0,C 180,E1 -22511.365,E2 -22511.365} C_VEL
LIN {X 0,Y 179.574,Z 681.842,A -85,B 0,C 180,E1 -22515.901,E2 -22515.901} C_VEL
LIN {X 0,Y 181.625,Z 673.576,A -85,B 0,C 180,E1 -22520.382,E2 -22520.382} C_VEL
LIN {X 0,Y 184.511,Z 663.838,A -85,B 0,C 180,E1 -22524.772,E2 -22524.772} C_VEL
LIN {X 0,Y 188.175,Z 652.369,A -85,B 0,C 180,E1 -22529.048,E2 -22529.048} C_VEL
LIN {X 0,Y 192.093,Z 640.088,A -85,B 0,C 180,E1 -22532.866,E2 -22532.866} C_VEL
LIN {X 0,Y 196.436,Z 627.221,A -85,B 0,C 180,E1 -22536.182,E2 -22536.182} C_VEL
LIN {X 0,Y 200.758,Z 613.894,A -85,B 0,C 180,E1 -22539.061,E2 -22539.061} C_VEL
LIN {X 0,Y 204.514,Z 601.549,A -85,B 0,C 180,E1 -22541.286,E2 -22541.286} C_VEL
LIN {X 0,Y 204.519,Z 599.669,A -85,B 0,C 180,E1 -22541.685,E2 -22541.685} C_VEL
LIN {X 0,Y 201.284,Z 589.297,A -85,B 0,C 180,E1 -22544.293,E2 -22544.293} C_VEL
LIN {X 0,Y 205.485,Z 588.811,A -85,B 0,C 180,E1 -22545.911,E2 -22545.911} C_VEL
LIN {X 0,Y 210.075,Z 587.324,A -85,B 0,C 180,E1 -22547.393,E2 -22547.393} C_VEL
LIN {X 0,Y 210.952,Z 588.374,A -85,B 0,C 180,E1 -22547.866,E2 -22547.866} C_VEL
LIN {X 0,Y 214.346,Z 596.639,A -85,B 0,C 180,E1 -22550.273,E2 -22550.273} C_VEL
LIN {X 0,Y 217.372,Z 606.211,A -85,B 0,C 180,E1 -22552.807,E2 -22552.807} C_VEL
LIN {X 0,Y 219.046,Z 615.468,A -85,B 0,C 180,E1 -22554.971,E2 -22554.971} C_VEL
LIN {X 0,Y 220.264,Z 626.729,A -85,B 0,C 180,E1 -22557.549,E2 -22557.549} C_VEL
LIN {X 0,Y 215.295,Z 640.825,A -85,B 0,C 180,E1 -22559.602,E2 -22559.602} C_VEL
LIN {X 0,Y 210.286,Z 653.334,A -85,B 0,C 180,E1 -22561.829,E2 -22561.829} C_VEL
LIN {X 0,Y 204.797,Z 665.933,A -85,B 0,C 180,E1 -22564.596,E2 -22564.596} C_VEL
LIN {X 0,Y 199.446,Z 677.46,A -85,B 0,C 180,E1 -22567.738,E2 -22567.738} C_VEL
LIN {X 0,Y 193.853,Z 688.573,A -85,B 0,C 180,E1 -22571.503,E2 -22571.503} C_VEL
LIN {X 0,Y 189.603,Z 696.766,A -85,B 0,C 180,E1 -22574.959,E2 -22574.959} C_VEL
LIN {X 0,Y 185.502,Z 704.757,A -85,B 0,C 180,E1 -22579.078,E2 -22579.078} C_VEL
LIN {X 0,Y 182.187,Z 711.424,A -85,B 0,C 180,E1 -22583.352,E2 -22583.352} C_VEL
LIN {X 0,Y 179.101,Z 718.032,A -85,B 0,C 180,E1 -22588.873,E2 -22588.873} C_VEL
LIN {X 0,Y 177.227,Z 722.93,A -85,B 0,C 180,E1 -22594.546,E2 -22594.546} C_VEL
LIN {X 0,Y 176.374,Z 725.665,A -85,B 0,C 180,E1 -22599.169,E2 -22599.169} C_VEL
LIN {X 0,Y 176.058,Z 727.498,A -85,B 0,C 180,E1 -22603.855,E2 -22603.855} C_VEL
LIN {X 0,Y 176.24,Z 728.298,A -85,B 0,C 180,E1 -22608.601,E2 -22608.601} C_VEL
LIN {X 0,Y 177.224,Z 728.001,A -85,B 0,C 180,E1 -22614.201,E2 -22614.201} C_VEL
LIN {X 0,Y 178.49,Z 726.968,A -85,B 0,C 180,E1 -22618.193,E2 -22618.193} C_VEL
LIN {X 0,Y 180.855,Z 724.696,A -85,B 0,C 180,E1 -22622.956,E2 -22622.956} C_VEL
LIN {X 0,Y 184.135,Z 721.36,A -85,B 0,C 180,E1 -22627.635,E2 -22627.635} C_VEL
LIN {X 0,Y 188.431,Z 716.76,A -85,B 0,C 180,E1 -22632.168,E2 -22632.168} C_VEL
LIN {X 0,Y 193.759,Z 710.866,A -85,B 0,C 180,E1 -22636.501,E2 -22636.501} C_VEL
LIN {X 0,Y 200.574,Z 702.956,A -85,B 0,C 180,E1 -22640.896,E2 -22640.896} C_VEL
LIN {X 0,Y 207.291,Z 694.644,A -85,B 0,C 180,E1 -22644.454,E2 -22644.454} C_VEL
LIN {X 0,Y 214.243,Z 685.286,A -85,B 0,C 180,E1 -22647.635,E2 -22647.635} C_VEL
LIN {X 0,Y 221.83,Z 674.138,A -85,B 0,C 180,E1 -22650.599,E2 -22650.599} C_VEL
LIN {X 0,Y 228.725,Z 662.865,A -85,B 0,C 180,E1 -22653.004,E2 -22653.004} C_VEL
LIN {X 0,Y 235.706,Z 650.165,A -85,B 0,C 180,E1 -22655.183,E2 -22655.183} C_VEL
LIN {X 0,Y 239.651,Z 642.157,A -85,B 0,C 180,E1 -22656.338,E2 -22656.338} C_VEL
LIN {X 0,Y 239.68,Z 636.902,A -85,B 0,C 180,E1 -22658.045,E2 -22658.045} C_VEL
LIN {X 0,Y 238.723,Z 630.051,A -85,B 0,C 180,E1 -22660.68,E2 -22660.68} C_VEL
LIN {X 0,Y 237.2,Z 623.301,A -85,B 0,C 180,E1 -22663.651,E2 -22663.651} C_VEL
LIN {X 0,Y 235.222,Z 616.723,A -85,B 0,C 180,E1 -22667.05,E2 -22667.05} C_VEL
LIN {X 0,Y 233.291,Z 611.151,A -85,B 0,C 180,E1 -22670.462,E2 -22670.462} C_VEL
LIN {X 0,Y 231.955,Z 607.752,A -85,B 0,C 180,E1 -22673.038,E2 -22673.038} C_VEL
LIN {X 0,Y 230.436,Z 604.06,A -85,B 0,C 180,E1 -22676.502,E2 -22676.502} C_VEL
LIN {X 0,Y 228.9,Z 600.509,A -85,B 0,C 180,E1 -22681.759,E2 -22681.759} C_VEL
LIN {X 0,Y 228.646,Z 599.771,A -85,B 0,C 180,E1 -22683.524,E2 -22683.524} C_VEL
LIN {X 0,Y 228.375,Z 600.052,A -85,B 0,C 180,E1 -22688.85,E2 -22688.85} C_VEL
LIN {X 0,Y 229.015,Z 601.189,A -85,B 0,C 180,E1 -22692.404,E2 -22692.404} C_VEL
LIN {X 0,Y 229.578,Z 602.06,A -85,B 0,C 180,E1 -22694.175,E2 -22694.175} C_VEL
LIN {X 0,Y 232.523,Z 607.913,A -85,B 0,C 180,E1 -22700.458,E2 -22700.458} C_VEL
LIN {X 0,Y 233.985,Z 611.55,A -85,B 0,C 180,E1 -22702.983,E2 -22702.983} C_VEL
LIN {X 0,Y 235.855,Z 619.415,A -85,B 0,C 180,E1 -22706.633,E2 -22706.633} C_VEL
LIN {X 0,Y 237.831,Z 629.878,A -85,B 0,C 180,E1 -22710.646,E2 -22710.646} C_VEL
LIN {X 0,Y 238.498,Z 635.406,A -85,B 0,C 180,E1 -22712.451,E2 -22712.451} C_VEL
LIN {X 0,Y 238.539,Z 636.907,A -85,B 0,C 180,E1 -22712.865,E2 -22712.865} C_VEL
LIN {X 0,Y 236.227,Z 650.338,A -85,B 0,C 180,E1 -22715.679,E2 -22715.679} C_VEL
LIN {X 0,Y 232.41,Z 664.303,A -85,B 0,C 180,E1 -22718.518,E2 -22718.518} C_VEL
LIN {X 0,Y 231.731,Z 666.542,A -85,B 0,C 180,E1 -22719.003,E2 -22719.003} C_VEL
LIN {X 0,Y 224.201,Z 680.108,A -85,B 0,C 180,E1 -22721.212,E2 -22721.212} C_VEL
LIN {X 0,Y 216.655,Z 692.498,A -85,B 0,C 180,E1 -22723.804,E2 -22723.804} C_VEL
LIN {X 0,Y 209.584,Z 703.13,A -85,B 0,C 180,E1 -22726.577,E2 -22726.577} C_VEL
LIN {X 0,Y 202.06,Z 713.611,A -85,B 0,C 180,E1 -22730.049,E2 -22730.049} C_VEL
LIN {X 0,Y 195.684,Z 722.109,A -85,B 0,C 180,E1 -22733.662,E2 -22733.662} C_VEL
LIN {X 0,Y 194.528,Z 723.654,A -85,B 0,C 180,E1 -22734.396,E2 -22734.396} C_VEL
LIN {X 0,Y 191.837,Z 726.448,A -85,B 0,C 180,E1 -22735.719,E2 -22735.719} C_VEL
LIN {X 0,Y 185.981,Z 730.704,A -85,B 0,C 180,E1 -22737.779,E2 -22737.779} C_VEL
LIN {X 0,Y 180.336,Z 734.526,A -85,B 0,C 180,E1 -22740.034,E2 -22740.034} C_VEL
LIN {X 0,Y 178.042,Z 736.607,A -85,B 0,C 180,E1 -22741.64,E2 -22741.64} C_VEL
LIN {X 0,Y 174.267,Z 741.384,A -85,B 0,C 180,E1 -22746.219,E2 -22746.219} C_VEL
LIN {X 0,Y 171.644,Z 744.97,A -85,B 0,C 180,E1 -22750.882,E2 -22750.882} C_VEL
LIN {X 0,Y 169.919,Z 747.637,A -85,B 0,C 180,E1 -22755.634,E2 -22755.634} C_VEL
LIN {X 0,Y 169.215,Z 749.272,A -85,B 0,C 180,E1 -22760.44,E2 -22760.44} C_VEL
LIN {X 0,Y 169.321,Z 750.022,A -85,B 0,C 180,E1 -22765.241,E2 -22765.241} C_VEL
LIN {X 0,Y 169.541,Z 749.697,A -85,B 0,C 180,E1 -22770.003,E2 -22770.003} C_VEL
LIN {X 0,Y 169.498,Z 749.174,A -85,B 0,C 180,E1 -22772.379,E2 -22772.379} C_VEL
LIN {X 0,Y 169.412,Z 748.117,A -85,B 0,C 180,E1 -22775.37,E2 -22775.37} C_VEL
LIN {X 0,Y 169.335,Z 745.89,A -85,B 0,C 180,E1 -22779.559,E2 -22779.559} C_VEL
LIN {X 0,Y 170.034,Z 742.406,A -85,B 0,C 180,E1 -22784.361,E2 -22784.361} C_VEL
LIN {X 0,Y 171.924,Z 736.847,A -85,B 0,C 180,E1 -22789.917,E2 -22789.917} C_VEL
LIN {X 0,Y 173.703,Z 732.755,A -85,B 0,C 180,E1 -22793.236,E2 -22793.236} C_VEL
LIN {X 0,Y 179.897,Z 727.685,A -85,B 0,C 180,E1 -22800.524,E2 -22800.524} C_VEL
LIN {X 0,Y 188.334,Z 721.634,A -85,B 0,C 180,E1 -22806.662,E2 -22806.662} C_VEL
LIN {X 0,Y 200.337,Z 713.824,A -85,B 0,C 180,E1 -22812.55,E2 -22812.55} C_VEL
LIN {X 0,Y 212.156,Z 706.525,A -85,B 0,C 180,E1 -22816.787,E2 -22816.787} C_VEL
LIN {X 0,Y 218.13,Z 702.914,A -85,B 0,C 180,E1 -22818.489,E2 -22818.489} C_VEL
LIN {X 0,Y 218.761,Z 702.392,A -85,B 0,C 180,E1 -22818.973,E2 -22818.973} C_VEL
LIN {X 0,Y 208.082,Z 705.728,A -85,B 0,C 180,E1 -22822.559,E2 -22822.559} C_VEL
LIN {X 0,Y 196.605,Z 708.695,A -85,B 0,C 180,E1 -22827.576,E2 -22827.576} C_VEL
LIN {X 0,Y 187.151,Z 710.381,A -85,B 0,C 180,E1 -22833.217,E2 -22833.217} C_VEL
LIN {X 0,Y 179.858,Z 710.628,A -85,B 0,C 180,E1 -22839.411,E2 -22839.411} C_VEL
LIN {X 0,Y 174.882,Z 709.296,A -85,B 0,C 180,E1 -22846.048,E2 -22846.048} C_VEL
LIN {X 0,Y 172.683,Z 707.47,A -85,B 0,C 180,E1 -22850.632,E2 -22850.632} C_VEL
LIN {X 0,Y 171.102,Z 704.916,A -85,B 0,C 180,E1 -22855.289,E2 -22855.289} C_VEL
LIN {X 0,Y 170.359,Z 700.44,A -85,B 0,C 180,E1 -22861.183,E2 -22861.183} C_VEL
LIN {X 0,Y 170.559,Z 695.774,A -85,B 0,C 180,E1 -22865.914,E2 -22865.914} C_VEL
LIN {X 0,Y 171.099,Z 690.126,A -85,B 0,C 180,E1 -22870.653,E2 -22870.653} C_VEL
LIN {X 0,Y 172.278,Z 683.279,A -85,B 0,C 180,E1 -22875.378,E2 -22875.378} C_VEL
LIN {X 0,Y 174.295,Z 675.11,A -85,B 0,C 180,E1 -22880.045,E2 -22880.045} C_VEL
LIN {X 0,Y 177.127,Z 665.515,A -85,B 0,C 180,E1 -22884.621,E2 -22884.621} C_VEL
LIN {X 0,Y 180.78,Z 654.27,A -85,B 0,C 180,E1 -22889.076,E2 -22889.076} C_VEL
LIN {X 0,Y 184.442,Z 643.277,A -85,B 0,C 180,E1 -22892.711,E2 -22892.711} C_VEL
LIN {X 0,Y 189.514,Z 628.449,A -85,B 0,C 180,E1 -22896.727,E2 -22896.727} C_VEL
LIN {X 0,Y 194.334,Z 613.968,A -85,B 0,C 180,E1 -22899.936,E2 -22899.936} C_VEL
LIN {X 0,Y 197.92,Z 602.736,A -85,B 0,C 180,E1 -22902.017,E2 -22902.017} C_VEL
LIN {X 0,Y 197.599,Z 600.7,A -85,B 0,C 180,E1 -22902.515,E2 -22902.515} C_VEL
LIN {X 0,Y 196.464,Z 596.869,A -85,B 0,C 180,E1 -22903.584,E2 -22903.584} C_VEL
LIN {X 0,Y 197.021,Z 597.206,A -85,B 0,C 180,E1 -22903.892,E2 -22903.892} C_VEL
LIN {X 0,Y 199.369,Z 596.899,A -85,B 0,C 180,E1 -22904.833,E2 -22904.833} C_VEL
LIN {X 0,Y 206.126,Z 594.849,A -85,B 0,C 180,E1 -22907.143,E2 -22907.143} C_VEL
LIN {X 0,Y 207.924,Z 596.359,A -85,B 0,C 180,E1 -22908.042,E2 -22908.042} C_VEL
LIN {X 0,Y 211.098,Z 605.606,A -85,B 0,C 180,E1 -22910.759,E2 -22910.759} C_VEL
LIN {X 0,Y 212.911,Z 613.096,A -85,B 0,C 180,E1 -22912.74,E2 -22912.74} C_VEL
LIN {X 0,Y 214.209,Z 624.165,A -85,B 0,C 180,E1 -22915.412,E2 -22915.412} C_VEL
LIN {X 0,Y 214.53,Z 628.481,A -85,B 0,C 180,E1 -22916.437,E2 -22916.437} C_VEL
LIN {X 0,Y 209.262,Z 642.943,A -85,B 0,C 180,E1 -22918.628,E2 -22918.628} C_VEL
LIN {X 0,Y 204.106,Z 655.168,A -85,B 0,C 180,E1 -22920.896,E2 -22920.896} C_VEL
LIN {X 0,Y 198.484,Z 667.53,A -85,B 0,C 180,E1 -22923.728,E2 -22923.728} C_VEL
LIN {X 0,Y 192.955,Z 678.872,A -85,B 0,C 180,E1 -22926.947,E2 -22926.947} C_VEL
LIN {X 0,Y 187.138,Z 689.852,A -85,B 0,C 180,E1 -22930.814,E2 -22930.814} C_VEL
LIN {X 0,Y 182.805,Z 697.94,A -85,B 0,C 180,E1 -22934.386,E2 -22934.386} C_VEL
LIN {X 0,Y 178.566,Z 705.796,A -85,B 0,C 180,E1 -22938.648,E2 -22938.648} C_VEL
LIN {X 0,Y 175.136,Z 712.359,A -85,B 0,C 180,E1 -22943.083,E2 -22943.083} C_VEL
LIN {X 0,Y 172.516,Z 717.666,A -85,B 0,C 180,E1 -22947.663,E2 -22947.663} C_VEL
LIN {X 0,Y 170.74,Z 721.888,A -85,B 0,C 180,E1 -22952.357,E2 -22952.357} C_VEL
LIN {X 0,Y 169.606,Z 725.11,A -85,B 0,C 180,E1 -22957.138,E2 -22957.138} C_VEL
LIN {X 0,Y 169.027,Z 727.288,A -85,B 0,C 180,E1 -22961.996,E2 -22961.996} C_VEL
LIN {X 0,Y 169.069,Z 728.581,A -85,B 0,C 180,E1 -22967.04,E2 -22967.04} C_VEL
LIN {X 0,Y 169.575,Z 728.781,A -85,B 0,C 180,E1 -22971.898,E2 -22971.898} C_VEL
LIN {X 0,Y 170.874,Z 728.05,A -85,B 0,C 180,E1 -22976.896,E2 -22976.896} C_VEL
LIN {X 0,Y 173.087,Z 726.24,A -85,B 0,C 180,E1 -22981.857,E2 -22981.857} C_VEL
LIN {X 0,Y 176.547,Z 722.974,A -85,B 0,C 180,E1 -22987.233,E2 -22987.233} C_VEL
LIN {X 0,Y 181.538,Z 718.054,A -85,B 0,C 180,E1 -22992.644,E2 -22992.644} C_VEL
LIN {X 0,Y 187.799,Z 711.602,A -85,B 0,C 180,E1 -22997.652,E2 -22997.652} C_VEL
LIN {X 0,Y 193.451,Z 705.492,A -85,B 0,C 180,E1 -23001.276,E2 -23001.276} C_VEL
LIN {X 0,Y 200.948,Z 696.73,A -85,B 0,C 180,E1 -23005.27,E2 -23005.27} C_VEL
LIN {X 0,Y 208.081,Z 687.614,A -85,B 0,C 180,E1 -23008.515,E2 -23008.515} C_VEL
LIN {X 0,Y 215.876,Z 676.864,A -85,B 0,C 180,E1 -23011.517,E2 -23011.517} C_VEL
LIN {X 0,Y 223.222,Z 665.557,A -85,B 0,C 180,E1 -23014.051,E2 -23014.051} C_VEL
LIN {X 0,Y 230.37,Z 653.325,A -85,B 0,C 180,E1 -23016.231,E2 -23016.231} C_VEL
LIN {X 0,Y 234.336,Z 645.783,A -85,B 0,C 180,E1 -23017.362,E2 -23017.362} C_VEL
LIN {X 0,Y 234.852,Z 644.058,A -85,B 0,C 180,E1 -23017.736,E2 -23017.736} C_VEL
LIN {X 0,Y 234.653,Z 638.276,A -85,B 0,C 180,E1 -23019.898,E2 -23019.898} C_VEL
LIN {X 0,Y 233.8,Z 632.146,A -85,B 0,C 180,E1 -23022.506,E2 -23022.506} C_VEL
LIN {X 0,Y 232.229,Z 625.148,A -85,B 0,C 180,E1 -23025.988,E2 -23025.988} C_VEL
LIN {X 0,Y 230.554,Z 619.281,A -85,B 0,C 180,E1 -23029.461,E2 -23029.461} C_VEL
LIN {X 0,Y 228.974,Z 614.536,A -85,B 0,C 180,E1 -23032.947,E2 -23032.947} C_VEL
LIN {X 0,Y 227.711,Z 610.788,A -85,B 0,C 180,E1 -23036.46,E2 -23036.46} C_VEL
LIN {X 0,Y 226.347,Z 607.196,A -85,B 0,C 180,E1 -23041.779,E2 -23041.779} C_VEL
LIN {X 0,Y 226.168,Z 606.44,A -85,B 0,C 180,E1 -23043.562,E2 -23043.562} C_VEL
LIN {X 0,Y 225.973,Z 606.746,A -85,B 0,C 180,E1 -23048.945,E2 -23048.945} C_VEL
LIN {X 0,Y 226.612,Z 607.94,A -85,B 0,C 180,E1 -23052.538,E2 -23052.538} C_VEL
LIN {X 0,Y 227.112,Z 608.969,A -85,B 0,C 180,E1 -23054.332,E2 -23054.332} C_VEL
LIN {X 0,Y 229.923,Z 614.904,A -85,B 0,C 180,E1 -23060.699,E2 -23060.699} C_VEL
LIN {X 0,Y 230.785,Z 617.402,A -85,B 0,C 180,E1 -23062.374,E2 -23062.374} C_VEL
LIN {X 0,Y 232.113,Z 624.469,A -85,B 0,C 180,E1 -23065.794,E2 -23065.794} C_VEL
LIN {X 0,Y 233.597,Z 634.375,A -85,B 0,C 180,E1 -23069.761,E2 -23069.761} C_VEL
LIN {X 0,Y 234.051,Z 639.966,A -85,B 0,C 180,E1 -23071.685,E2 -23071.685} C_VEL
LIN {X 0,Y 232.461,Z 648.656,A -85,B 0,C 180,E1 -23073.616,E2 -23073.616} C_VEL
LIN {X 0,Y 230.297,Z 657.232,A -85,B 0,C 180,E1 -23075.437,E2 -23075.437} C_VEL
LIN {X 0,Y 226.774,Z 668.274,A -85,B 0,C 180,E1 -23077.793,E2 -23077.793} C_VEL
LIN {X 0,Y 219.596,Z 680.503,A -85,B 0,C 180,E1 -23079.82,E2 -23079.82} C_VEL
LIN {X 0,Y 211.785,Z 692.739,A -85,B 0,C 180,E1 -23082.412,E2 -23082.412} C_VEL
LIN {X 0,Y 204.452,Z 703.252,A -85,B 0,C 180,E1 -23085.2,E2 -23085.2} C_VEL
LIN {X 0,Y 196.99,Z 713.174,A -85,B 0,C 180,E1 -23088.521,E2 -23088.521} C_VEL
LIN {X 0,Y 189.949,Z 722.08,A -85,B 0,C 180,E1 -23092.378,E2 -23092.378} C_VEL
LIN {X 0,Y 184.012,Z 729.328,A -85,B 0,C 180,E1 -23096.375,E2 -23096.375} C_VEL
LIN {X 0,Y 179.032,Z 735.408,A -85,B 0,C 180,E1 -23100.617,E2 -23100.617} C_VEL
LIN {X 0,Y 178.042,Z 736.607,A -85,B 0,C 180,E1 -23101.64,E2 -23101.64} C_VEL
LIN {X 0,Y 175.875,Z 738.604,A -85,B 0,C 180,E1 -23103.304,E2 -23103.304} C_VEL
LIN {X 0,Y 170.87,Z 741.467,A -85,B 0,C 180,E1 -23105.969,E2 -23105.969} C_VEL
LIN {X 0,Y 166.963,Z 743.404,A -85,B 0,C 180,E1 -23108.223,E2 -23108.223} C_VEL
LIN {X 0,Y 164.913,Z 744.673,A -85,B 0,C 180,E1 -23110.089,E2 -23110.089} C_VEL
LIN {X 0,Y 164.518,Z 745.056,A -85,B 0,C 180,E1 -23110.746,E2 -23110.746} C_VEL
LIN {X 0,Y 162.977,Z 747.285,A -85,B 0,C 180,E1 -23115.008,E2 -23115.008} C_VEL
LIN {X 0,Y 162.143,Z 748.862,A -85,B 0,C 180,E1 -23120.019,E2 -23120.019} C_VEL
LIN {X 0,Y 162.25,Z 749.582,A -85,B 0,C 180,E1 -23125.033,E2 -23125.033} C_VEL
LIN {X 0,Y 162.474,Z 749.2,A -85,B 0,C 180,E1 -23130.003,E2 -23130.003} C_VEL
LIN {X 0,Y 162.34,Z 747.837,A -85,B 0,C 180,E1 -23134.97,E2 -23134.97} C_VEL
LIN {X 0,Y 162.284,Z 745.291,A -85,B 0,C 180,E1 -23139.978,E2 -23139.978} C_VEL
LIN {X 0,Y 163.091,Z 741.736,A -85,B 0,C 180,E1 -23144.987,E2 -23144.987} C_VEL
LIN {X 0,Y 164.962,Z 736.521,A -85,B 0,C 180,E1 -23150.403,E2 -23150.403} C_VEL
LIN {X 0,Y 167.072,Z 732.15,A -85,B 0,C 180,E1 -23154.216,E2 -23154.216} C_VEL
LIN {X 0,Y 171.341,Z 729.081,A -85,B 0,C 180,E1 -23159.489,E2 -23159.489} C_VEL
LIN {X 0,Y 179.383,Z 723.812,A -85,B 0,C 180,E1 -23165.995,E2 -23165.995} C_VEL
LIN {X 0,Y 190.001,Z 717.51,A -85,B 0,C 180,E1 -23171.747,E2 -23171.747} C_VEL
LIN {X 0,Y 205.043,Z 709.029,A -85,B 0,C 180,E1 -23177.473,E2 -23177.473} C_VEL
LIN {X 0,Y 208.755,Z 706.949,A -85,B 0,C 180,E1 -23178.577,E2 -23178.577} C_VEL
LIN {X 0,Y 209.468,Z 706.391,A -85,B 0,C 180,E1 -23179.15,E2 -23179.15} C_VEL
LIN {X 0,Y 198.601,Z 709.088,A -85,B 0,C 180,E1 -23183.017,E2 -23183.017} C_VEL
LIN {X 0,Y 187.376,Z 711.18,A -85,B 0,C 180,E1 -23188.326,E2 -23188.326} C_VEL
LIN {X 0,Y 178.225,Z 712.004,A -85,B 0,C 180,E1 -23194.294,E2 -23194.294} C_VEL
LIN {X 0,Y 171.269,Z 711.393,A -85,B 0,C 180,E1 -23200.837,E2 -23200.837} C_VEL
LIN {X 0,Y 166.789,Z 709.169,A -85,B 0,C 180,E1 -23207.839,E2 -23207.839} C_VEL
LIN {X 0,Y 164.781,Z 706.755,A -85,B 0,C 180,E1 -23212.65,E2 -23212.65} C_VEL
LIN {X 0,Y 163.564,Z 703.561,A -85,B 0,C 180,E1 -23217.538,E2 -23217.538} C_VEL
LIN {X 0,Y 163.334,Z 698.275,A -85,B 0,C 180,E1 -23223.702,E2 -23223.702} C_VEL
LIN {X 0,Y 163.817,Z 692.003,A -85,B 0,C 180,E1 -23229.399,E2 -23229.399} C_VEL
LIN {X 0,Y 164.96,Z 684.625,A -85,B 0,C 180,E1 -23234.812,E2 -23234.812} C_VEL
LIN {X 0,Y 167.224,Z 675.505,A -85,B 0,C 180,E1 -23240.288,E2 -23240.288} C_VEL
LIN {X 0,Y 170.151,Z 665.824,A -85,B 0,C 180,E1 -23245.049,E2 -23245.049} C_VEL
LIN {X 0,Y 173.92,Z 654.464,A -85,B 0,C 180,E1 -23249.672,E2 -23249.672} C_VEL
LIN {X 0,Y 177.89,Z 642.944,A -85,B 0,C 180,E1 -23253.582,E2 -23253.582} C_VEL
LIN {X 0,Y 182.607,Z 629.669,A -85,B 0,C 180,E1 -23257.314,E2 -23257.314} C_VEL
LIN {X 0,Y 187.543,Z 615.244,A -85,B 0,C 180,E1 -23260.627,E2 -23260.627} C_VEL
LIN {X 0,Y 191.309,Z 604.178,A -85,B 0,C 180,E1 -23262.802,E2 -23262.802} C_VEL
LIN {X 0,Y 193.174,Z 604.512,A -85,B 0,C 180,E1 -23263.731,E2 -23263.731} C_VEL
LIN {X 0,Y 202.037,Z 602.151,A -85,B 0,C 180,E1 -23266.93,E2 -23266.93} C_VEL
LIN {X 0,Y 204.041,Z 602.661,A -85,B 0,C 180,E1 -23267.779,E2 -23267.779} C_VEL
LIN {X 0,Y 207.07,Z 613.174,A -85,B 0,C 180,E1 -23270.907,E2 -23270.907} C_VEL
LIN {X 0,Y 208.292,Z 621.869,A -85,B 0,C 180,E1 -23273.176,E2 -23273.176} C_VEL
LIN {X 0,Y 208.831,Z 629.507,A -85,B 0,C 180,E1 -23275.1,E2 -23275.1} C_VEL
LIN {X 0,Y 208.763,Z 630.966,A -85,B 0,C 180,E1 -23275.442,E2 -23275.442} C_VEL
LIN {X 0,Y 203.794,Z 643.777,A -85,B 0,C 180,E1 -23277.393,E2 -23277.393} C_VEL
LIN {X 0,Y 197.985,Z 656.99,A -85,B 0,C 180,E1 -23279.905,E2 -23279.905} C_VEL
LIN {X 0,Y 192.185,Z 669.133,A -85,B 0,C 180,E1 -23282.797,E2 -23282.797} C_VEL
LIN {X 0,Y 186.501,Z 680.284,A -85,B 0,C 180,E1 -23286.101,E2 -23286.101} C_VEL
LIN {X 0,Y 181.21,Z 689.89,A -85,B 0,C 180,E1 -23289.568,E2 -23289.568} C_VEL
LIN {X 0,Y 176.589,Z 698.028,A -85,B 0,C 180,E1 -23293.227,E2 -23293.227} C_VEL
LIN {X 0,Y 172.661,Z 705.057,A -85,B 0,C 180,E1 -23297.061,E2 -23297.061} C_VEL
LIN {X 0,Y 168.905,Z 711.793,A -85,B 0,C 180,E1 -23301.624,E2 -23301.624} C_VEL
LIN {X 0,Y 165.984,Z 717.296,A -85,B 0,C 180,E1 -23306.356,E2 -23306.356} C_VEL
LIN {X 0,Y 164.368,Z 720.708,A -85,B 0,C 180,E1 -23309.997,E2 -23309.997} C_VEL
LIN {X 0,Y 162.964,Z 724.332,A -85,B 0,C 180,E1 -23314.945,E2 -23314.945} C_VEL
LIN {X 0,Y 162.087,Z 726.96,A -85,B 0,C 180,E1 -23319.985,E2 -23319.985} C_VEL
LIN {X 0,Y 161.891,Z 728.584,A -85,B 0,C 180,E1 -23325.095,E2 -23325.095} C_VEL
LIN {X 0,Y 162.22,Z 729.292,A -85,B 0,C 180,E1 -23330.276,E2 -23330.276} C_VEL
LIN {X 0,Y 163.355,Z 728.923,A -85,B 0,C 180,E1 -23335.479,E2 -23335.479} C_VEL
LIN {X 0,Y 165.307,Z 727.599,A -85,B 0,C 180,E1 -23340.672,E2 -23340.672} C_VEL
LIN {X 0,Y 168.241,Z 725.146,A -85,B 0,C 180,E1 -23345.787,E2 -23345.787} C_VEL
LIN {X 0,Y 172.256,Z 721.571,A -85,B 0,C 180,E1 -23350.749,E2 -23350.749} C_VEL
LIN {X 0,Y 177.365,Z 716.826,A -85,B 0,C 180,E1 -23355.495,E2 -23355.495} C_VEL
LIN {X 0,Y 183.54,Z 710.701,A -85,B 0,C 180,E1 -23359.976,E2 -23359.976} C_VEL
LIN {X 0,Y 190.69,Z 703.121,A -85,B 0,C 180,E1 -23364.172,E2 -23364.172} C_VEL
LIN {X 0,Y 198.755,Z 693.891,A -85,B 0,C 180,E1 -23368.059,E2 -23368.059} C_VEL
LIN {X 0,Y 206.459,Z 684.23,A -85,B 0,C 180,E1 -23371.223,E2 -23371.223} C_VEL
LIN {X 0,Y 213.535,Z 674.545,A -85,B 0,C 180,E1 -23373.744,E2 -23373.744} C_VEL
LIN {X 0,Y 220.984,Z 663.125,A -85,B 0,C 180,E1 -23376.135,E2 -23376.135} C_VEL
LIN {X 0,Y 227.786,Z 651.534,A -85,B 0,C 180,E1 -23378.089,E2 -23378.089} C_VEL
LIN {X 0,Y 229.646,Z 648.111,A -85,B 0,C 180,E1 -23378.594,E2 -23378.594} C_VEL
LIN {X 0,Y 229.981,Z 646.831,A -85,B 0,C 180,E1 -23378.956,E2 -23378.956} C_VEL
LIN {X 0,Y 229.736,Z 640.657,A -85,B 0,C 180,E1 -23381.495,E2 -23381.495} C_VEL
LIN {X 0,Y 229.07,Z 635.34,A -85,B 0,C 180,E1 -23383.97,E2 -23383.97} C_VEL
LIN {X 0,Y 228.129,Z 630.352,A -85,B 0,C 180,E1 -23386.64,E2 -23386.64} C_VEL
LIN {X 0,Y 226.819,Z 624.681,A -85,B 0,C 180,E1 -23390.187,E2 -23390.187} C_VEL
LIN {X 0,Y 225.793,Z 621.182,A -85,B 0,C 180,E1 -23392.847,E2 -23392.847} C_VEL
LIN {X 0,Y 224.708,Z 617.42,A -85,B 0,C 180,E1 -23396.413,E2 -23396.413} C_VEL
LIN {X 0,Y 223.803,Z 614.86,A -85,B 0,C 180,E1 -23399.999,E2 -23399.999} C_VEL
